LIN {X 0,Y 450.056,Z 1227.02,A -85,B 0,C 180,E1 22125.46,E2 22125.46} C_VEL
LIN {X 0,Y 451.314,Z 1216.532,A -85,B 0,C 180,E1 22122.995,E2 22122.995} C_VEL
LIN {X 0,Y 453.016,Z 1203.981,A -85,B 0,C 180,E1 22120.532,E2 22120.532} C_VEL
LIN {X 0,Y 454.944,Z 1190.743,A -85,B 0,C 180,E1 22118.331,E2 22118.331} C_VEL
LIN {X 0,Y 457.28,Z 1175.115,A -85,B 0,C 180,E1 22116.139,E2 22116.139} C_VEL
LIN {X 0,Y 459.71,Z 1158.959,A -85,B 0,C 180,E1 22114.214,E2 22114.214} C_VEL
LIN {X 0,Y 462.395,Z 1140.754,A -85,B 0,C 180,E1 22112.365,E2 22112.365} C_VEL
LIN {X 0,Y 464.992,Z 1122.424,A -85,B 0,C 180,E1 22110.782,E2 22110.782} C_VEL
LIN {X 0,Y 467.714,Z 1101.621,A -85,B 0,C 180,E1 22109.273,E2 22109.273} C_VEL
LIN {X 0,Y 470.333,Z 1079.541,A -85,B 0,C 180,E1 22107.966,E2 22107.966} C_VEL
LIN {X 0,Y 472.543,Z 1057.663,A -85,B 0,C 180,E1 22106.923,E2 22106.923} C_VEL
LIN {X 0,Y 474.461,Z 1035.079,A -85,B 0,C 180,E1 22106.08,E2 22106.08} C_VEL
LIN {X 0,Y 476.032,Z 1011.751,A -85,B 0,C 180,E1 22105.437,E2 22105.437} C_VEL
LIN {X 0,Y 488.439,Z 758.371,A -85,B 0,C 180,E1 22100.652,E2 22100.652} C_VEL
LIN {X 0,Y 471.567,Z 725.378,A -85,B 0,C 180,E1 22098.484,E2 22098.484} C_VEL
LIN {X 0,Y 462.172,Z 707.758,A -85,B 0,C 180,E1 22097.175,E2 22097.175} C_VEL
LIN {X 0,Y 454.225,Z 686.767,A -85,B 0,C 180,E1 22094.078,E2 22094.078} C_VEL
LIN {X 0,Y 450.292,Z 676.573,A -85,B 0,C 180,E1 22092.505,E2 22092.505} C_VEL
LIN {X 0,Y 450.29,Z 676.583,A -85,B 0,C 180,E1 22088.793,E2 22088.793} C_VEL
LIN {X 0,Y 450.29,Z 676.576,A -85,B 0,C 180,E1 22084.977,E2 22084.977} C_VEL
LIN {X 0,Y 450.301,Z 676.568,A -85,B 0,C 180,E1 22081.252,E2 22081.252} C_VEL
LIN {X 0,Y 450.289,Z 676.577,A -85,B 0,C 180,E1 22077.51,E2 22077.51} C_VEL
LIN {X 0,Y 450.301,Z 676.576,A -85,B 0,C 180,E1 22073.816,E2 22073.816} C_VEL
LIN {X 0,Y 450.302,Z 676.577,A -85,B 0,C 180,E1 22069.998,E2 22069.998} C_VEL
LIN {X 0,Y 450.288,Z 676.578,A -85,B 0,C 180,E1 22066.249,E2 22066.249} C_VEL
LIN {X 0,Y 450.3,Z 676.565,A -85,B 0,C 180,E1 22062.57,E2 22062.57} C_VEL
LIN {X 0,Y 450.284,Z 676.564,A -85,B 0,C 180,E1 22058.815,E2 22058.815} C_VEL
LIN {X 0,Y 450.291,Z 676.573,A -85,B 0,C 180,E1 22055.097,E2 22055.097} C_VEL
LIN {X 0,Y 450.29,Z 676.577,A -85,B 0,C 180,E1 22051.274,E2 22051.274} C_VEL
LIN {X 0,Y 450.289,Z 676.578,A -85,B 0,C 180,E1 22047.584,E2 22047.584} C_VEL
LIN {X 0,Y 450.296,Z 676.578,A -85,B 0,C 180,E1 22043.883,E2 22043.883} C_VEL
LIN {X 0,Y 450.289,Z 676.58,A -85,B 0,C 180,E1 22040.157,E2 22040.157} C_VEL
LIN {X 0,Y 450.288,Z 676.568,A -85,B 0,C 180,E1 22038.847,E2 22038.847} C_VEL
LIN {X 0,Y 449.316,Z 676.698,A -85,B 0,C 180,E1 22037.866,E2 22037.866} C_VEL
LIN {X 0,Y 442.815,Z 677.506,A -85,B 0,C 180,E1 22035.035,E2 22035.035} C_VEL
LIN {X 0,Y 442.36,Z 677.568,A -85,B 0,C 180,E1 22034.387,E2 22034.387} C_VEL
LIN {X 0,Y 442.357,Z 677.564,A -85,B 0,C 180,E1 22030.595,E2 22030.595} C_VEL
LIN {X 0,Y 442.355,Z 677.564,A -85,B 0,C 180,E1 22026.842,E2 22026.842} C_VEL
LIN {X 0,Y 442.362,Z 677.562,A -85,B 0,C 180,E1 22023.126,E2 22023.126} C_VEL
LIN {X 0,Y 442.352,Z 677.568,A -85,B 0,C 180,E1 22019.282,E2 22019.282} C_VEL
LIN {X 0,Y 442.377,Z 677.726,A -85,B 0,C 180,E1 22019.086,E2 22019.086} C_VEL
LIN {X 0,Y 443.743,Z 681.144,A -85,B 0,C 180,E1 22018.485,E2 22018.485} C_VEL
LIN {X 0,Y 450.868,Z 697.83,A -85,B 0,C 180,E1 22015.565,E2 22015.565} C_VEL
LIN {X 0,Y 458.461,Z 716.626,A -85,B 0,C 180,E1 22012.522,E2 22012.522} C_VEL
LIN {X 0,Y 466.093,Z 737.615,A -85,B 0,C 180,E1 22009.414,E2 22009.414} C_VEL
LIN {X 0,Y 472.641,Z 757.701,A -85,B 0,C 180,E1 22006.671,E2 22006.671} C_VEL
LIN {X 0,Y 467.674,Z 797.424,A -85,B 0,C 180,E1 22003.002,E2 22003.002} C_VEL
LIN {X 0,Y 462.803,Z 839.96,A -85,B 0,C 180,E1 21999.115,E2 21999.115} C_VEL
LIN {X 0,Y 458.303,Z 884.233,A -85,B 0,C 180,E1 21995.105,E2 21995.105} C_VEL
LIN {X 0,Y 455.719,Z 913.64,A -85,B 0,C 180,E1 21992.499,E2 21992.499} C_VEL
LIN {X 0,Y 456.506,Z 925.556,A -85,B 0,C 180,E1 21992.153,E2 21992.153} C_VEL
LIN {X 0,Y 451.281,Z 1032.151,A -85,B 0,C 180,E1 21989.514,E2 21989.514} C_VEL
LIN {X 0,Y 450.142,Z 1064.631,A -85,B 0,C 180,E1 21988.597,E2 21988.597} C_VEL
LIN {X 0,Y 449.375,Z 1081.923,A -85,B 0,C 180,E1 21987.857,E2 21987.857} C_VEL
LIN {X 0,Y 448.364,Z 1098.592,A -85,B 0,C 180,E1 21986.876,E2 21986.876} C_VEL
LIN {X 0,Y 447.221,Z 1113.837,A -85,B 0,C 180,E1 21985.713,E2 21985.713} C_VEL
LIN {X 0,Y 446.029,Z 1128.635,A -85,B 0,C 180,E1 21984.291,E2 21984.291} C_VEL
LIN {X 0,Y 444.836,Z 1141.996,A -85,B 0,C 180,E1 21982.674,E2 21982.674} C_VEL
LIN {X 0,Y 443.812,Z 1153.261,A -85,B 0,C 180,E1 21980.991,E2 21980.991} C_VEL
LIN {X 0,Y 442.868,Z 1164.02,A -85,B 0,C 180,E1 21978.973,E2 21978.973} C_VEL
LIN {X 0,Y 442.222,Z 1172.371,A -85,B 0,C 180,E1 21976.958,E2 21976.958} C_VEL
LIN {X 0,Y 441.818,Z 1178.872,A -85,B 0,C 180,E1 21974.915,E2 21974.915} C_VEL
LIN {X 0,Y 441.638,Z 1183.6,A -85,B 0,C 180,E1 21972.819,E2 21972.819} C_VEL
LIN {X 0,Y 441.67,Z 1186.819,A -85,B 0,C 180,E1 21970.566,E2 21970.566} C_VEL
LIN {X 0,Y 441.926,Z 1188.049,A -85,B 0,C 180,E1 21968.326,E2 21968.326} C_VEL
LIN {X 0,Y 442.395,Z 1187.557,A -85,B 0,C 180,E1 21966.228,E2 21966.228} C_VEL
LIN {X 0,Y 443.192,Z 1185.187,A -85,B 0,C 180,E1 21964.011,E2 21964.011} C_VEL
LIN {X 0,Y 444.276,Z 1181.299,A -85,B 0,C 180,E1 21961.935,E2 21961.935} C_VEL
LIN {X 0,Y 445.808,Z 1175.142,A -85,B 0,C 180,E1 21959.743,E2 21959.743} C_VEL
LIN {X 0,Y 447.557,Z 1167.915,A -85,B 0,C 180,E1 21957.823,E2 21957.823} C_VEL
LIN {X 0,Y 449.67,Z 1158.688,A -85,B 0,C 180,E1 21955.92,E2 21955.92} C_VEL
LIN {X 0,Y 451.78,Z 1148.729,A -85,B 0,C 180,E1 21954.284,E2 21954.284} C_VEL
LIN {X 0,Y 454.277,Z 1136.036,A -85,B 0,C 180,E1 21952.602,E2 21952.602} C_VEL
LIN {X 0,Y 456.731,Z 1121.995,A -85,B 0,C 180,E1 21951.121,E2 21951.121} C_VEL
LIN {X 0,Y 458.851,Z 1108.131,A -85,B 0,C 180,E1 21949.96,E2 21949.96} C_VEL
LIN {X 0,Y 460.981,Z 1091.626,A -85,B 0,C 180,E1 21948.869,E2 21948.869} C_VEL
LIN {X 0,Y 462.692,Z 1074.772,A -85,B 0,C 180,E1 21948.026,E2 21948.026} C_VEL
LIN {X 0,Y 466.759,Z 1039.48,A -85,B 0,C 180,E1 21946.627,E2 21946.627} C_VEL
LIN {X 0,Y 474.203,Z 984.707,A -85,B 0,C 180,E1 21944.726,E2 21944.726} C_VEL
LIN {X 0,Y 479.772,Z 939.46,A -85,B 0,C 180,E1 21943.332,E2 21943.332} C_VEL
LIN {X 0,Y 479.663,Z 936.85,A -85,B 0,C 180,E1 21943.157,E2 21943.157} C_VEL
LIN {X 0,Y 489.104,Z 900.674,A -85,B 0,C 180,E1 21939.288,E2 21939.288} C_VEL
LIN {X 0,Y 499.739,Z 867.838,A -85,B 0,C 180,E1 21935.659,E2 21935.659} C_VEL
LIN {X 0,Y 511.957,Z 837.578,A -85,B 0,C 180,E1 21932.174,E2 21932.174} C_VEL
LIN {X 0,Y 521.645,Z 817.739,A -85,B 0,C 180,E1 21929.791,E2 21929.791} C_VEL
LIN {X 0,Y 522.316,Z 814.236,A -85,B 0,C 180,E1 21928.105,E2 21928.105} C_VEL
LIN {X 0,Y 522.83,Z 812.775,A -85,B 0,C 180,E1 21926.841,E2 21926.841} C_VEL
LIN {X 0,Y 523.839,Z 811.873,A -85,B 0,C 180,E1 21925.332,E2 21925.332} C_VEL
LIN {X 0,Y 523.786,Z 813.12,A -85,B 0,C 180,E1 21924.408,E2 21924.408} C_VEL
LIN {X 0,Y 511.159,Z 837.266,A -85,B 0,C 180,E1 21922.025,E2 21922.025} C_VEL
LIN {X 0,Y 502.911,Z 857.599,A -85,B 0,C 180,E1 21919.896,E2 21919.896} C_VEL
LIN {X 0,Y 497.203,Z 877.592,A -85,B 0,C 180,E1 21917.647,E2 21917.647} C_VEL
LIN {X 0,Y 494.543,Z 895.305,A -85,B 0,C 180,E1 21915.535,E2 21915.535} C_VEL
LIN {X 0,Y 494.336,Z 913.318,A -85,B 0,C 180,E1 21913.266,E2 21913.266} C_VEL
LIN {X 0,Y 496.692,Z 929.505,A -85,B 0,C 180,E1 21911.157,E2 21911.157} C_VEL
LIN {X 0,Y 501.231,Z 945.016,A -85,B 0,C 180,E1 21909.095,E2 21909.095} C_VEL
LIN {X 0,Y 488.403,Z 970.998,A -85,B 0,C 180,E1 21908.038,E2 21908.038} C_VEL
LIN {X 0,Y 478.774,Z 994.4,A -85,B 0,C 180,E1 21906.916,E2 21906.916} C_VEL
LIN {X 0,Y 474.737,Z 1026.804,A -85,B 0,C 180,E1 21906.44,E2 21906.44} C_VEL
LIN {X 0,Y 472.39,Z 1050.839,A -85,B 0,C 180,E1 21905.821,E2 21905.821} C_VEL
LIN {X 0,Y 469.098,Z 1076.984,A -85,B 0,C 180,E1 21904.909,E2 21904.909} C_VEL
LIN {X 0,Y 465.898,Z 1098.995,A -85,B 0,C 180,E1 21903.915,E2 21903.915} C_VEL
LIN {X 0,Y 462.099,Z 1123.392,A -85,B 0,C 180,E1 21902.525,E2 21902.525} C_VEL
LIN {X 0,Y 458.733,Z 1143.969,A -85,B 0,C 180,E1 21901.101,E2 21901.101} C_VEL
LIN {X 0,Y 453.603,Z 1177.436,A -85,B 0,C 180,E1 21898.359,E2 21898.359} C_VEL
LIN {X 0,Y 450.76,Z 1196.691,A -85,B 0,C 180,E1 21896.476,E2 21896.476} C_VEL
LIN {X 0,Y 448.232,Z 1213.866,A -85,B 0,C 180,E1 21894.474,E2 21894.474} C_VEL
LIN {X 0,Y 446.026,Z 1229.04,A -85,B 0,C 180,E1 21892.4,E2 21892.4} C_VEL
LIN {X 0,Y 444.101,Z 1243.186,A -85,B 0,C 180,E1 21890.136,E2 21890.136} C_VEL
LIN {X 0,Y 442.582,Z 1255.81,A -85,B 0,C 180,E1 21887.756,E2 21887.756} C_VEL
LIN {X 0,Y 441.424,Z 1266.903,A -85,B 0,C 180,E1 21885.232,E2 21885.232} C_VEL
LIN {X 0,Y 440.697,Z 1276.161,A -85,B 0,C 180,E1 21882.676,E2 21882.676} C_VEL
LIN {X 0,Y 440.308,Z 1283.784,A -85,B 0,C 180,E1 21880.068,E2 21880.068} C_VEL
LIN {X 0,Y 440.178,Z 1289.391,A -85,B 0,C 180,E1 21877.569,E2 21877.569} C_VEL
LIN {X 0,Y 440.187,Z 1293.587,A -85,B 0,C 180,E1 21874.95,E2 21874.95} C_VEL
LIN {X 0,Y 440.235,Z 1296.109,A -85,B 0,C 180,E1 21872.472,E2 21872.472} C_VEL
LIN {X 0,Y 440.268,Z 1297.032,A -85,B 0,C 180,E1 21869.998,E2 21869.998} C_VEL
LIN {X 0,Y 440.212,Z 1296.537,A -85,B 0,C 180,E1 21867.395,E2 21867.395} C_VEL
LIN {X 0,Y 440.144,Z 1294.495,A -85,B 0,C 180,E1 21864.915,E2 21864.915} C_VEL
LIN {X 0,Y 440.148,Z 1290.595,A -85,B 0,C 180,E1 21862.164,E2 21862.164} C_VEL
LIN {X 0,Y 440.341,Z 1285.146,A -85,B 0,C 180,E1 21859.491,E2 21859.491} C_VEL
LIN {X 0,Y 440.893,Z 1277.648,A -85,B 0,C 180,E1 21856.757,E2 21856.757} C_VEL
LIN {X 0,Y 441.861,Z 1268.533,A -85,B 0,C 180,E1 21854.1,E2 21854.1} C_VEL
LIN {X 0,Y 443.288,Z 1258.134,A -85,B 0,C 180,E1 21851.59,E2 21851.59} C_VEL
LIN {X 0,Y 445.269,Z 1245.64,A -85,B 0,C 180,E1 21849.079,E2 21849.079} C_VEL
LIN {X 0,Y 447.716,Z 1231.692,A -85,B 0,C 180,E1 21846.714,E2 21846.714} C_VEL
LIN {X 0,Y 450.8,Z 1215.453,A -85,B 0,C 180,E1 21844.371,E2 21844.371} C_VEL
LIN {X 0,Y 454.225,Z 1198.101,A -85,B 0,C 180,E1 21842.243,E2 21842.243} C_VEL
LIN {X 0,Y 457.98,Z 1179.391,A -85,B 0,C 180,E1 21840.289,E2 21840.289} C_VEL
LIN {X 0,Y 462.201,Z 1158.237,A -85,B 0,C 180,E1 21838.43,E2 21838.43} C_VEL
LIN {X 0,Y 466.546,Z 1136.041,A -85,B 0,C 180,E1 21836.797,E2 21836.797} C_VEL
LIN {X 0,Y 470.757,Z 1113.889,A -85,B 0,C 180,E1 21835.45,E2 21835.45} C_VEL
LIN {X 0,Y 475.07,Z 1090.125,A -85,B 0,C 180,E1 21834.262,E2 21834.262} C_VEL
LIN {X 0,Y 479.303,Z 1065.271,A -85,B 0,C 180,E1 21833.286,E2 21833.286} C_VEL
LIN {X 0,Y 483.325,Z 1037.764,A -85,B 0,C 180,E1 21832.445,E2 21832.445} C_VEL
LIN {X 0,Y 486.658,Z 1015.568,A -85,B 0,C 180,E1 21831.951,E2 21831.951} C_VEL
LIN {X 0,Y 492.888,Z 982.261,A -85,B 0,C 180,E1 21831.411,E2 21831.411} C_VEL
LIN {X 0,Y 499.024,Z 954.26,A -85,B 0,C 180,E1 21831.118,E2 21831.118} C_VEL
LIN {X 0,Y 501.49,Z 943.396,A -85,B 0,C 180,E1 21831.019,E2 21831.019} C_VEL
LIN {X 0,Y 498.054,Z 928.988,A -85,B 0,C 180,E1 21829.189,E2 21829.189} C_VEL
LIN {X 0,Y 497.038,Z 917.484,A -85,B 0,C 180,E1 21827.693,E2 21827.693} C_VEL
LIN {X 0,Y 497.581,Z 906.994,A -85,B 0,C 180,E1 21826.402,E2 21826.402} C_VEL
LIN {X 0,Y 499.538,Z 895.357,A -85,B 0,C 180,E1 21824.944,E2 21824.944} C_VEL
LIN {X 0,Y 502.528,Z 884.79,A -85,B 0,C 180,E1 21823.757,E2 21823.757} C_VEL
LIN {X 0,Y 506.992,Z 873.197,A -85,B 0,C 180,E1 21822.425,E2 21822.425} C_VEL
LIN {X 0,Y 510.787,Z 864.66,A -85,B 0,C 180,E1 21821.584,E2 21821.584} C_VEL
LIN {X 0,Y 498.036,Z 933.263,A -85,B 0,C 180,E1 21819.708,E2 21819.708} C_VEL
LIN {X 0,Y 488.405,Z 996.354,A -85,B 0,C 180,E1 21818.004,E2 21818.004} C_VEL
LIN {X 0,Y 483.779,Z 1031.006,A -85,B 0,C 180,E1 21817.02,E2 21817.02} C_VEL
LIN {X 0,Y 480.204,Z 1054.828,A -85,B 0,C 180,E1 21816.105,E2 21816.105} C_VEL
LIN {X 0,Y 476.468,Z 1077.16,A -85,B 0,C 180,E1 21815.027,E2 21815.027} C_VEL
LIN {X 0,Y 472.331,Z 1099.651,A -85,B 0,C 180,E1 21813.686,E2 21813.686} C_VEL
LIN {X 0,Y 468.084,Z 1121.13,A -85,B 0,C 180,E1 21812.134,E2 21812.134} C_VEL
LIN {X 0,Y 463.799,Z 1141.476,A -85,B 0,C 180,E1 21810.368,E2 21810.368} C_VEL
LIN {X 0,Y 459.71,Z 1160.043,A -85,B 0,C 180,E1 21808.446,E2 21808.446} C_VEL
LIN {X 0,Y 455.964,Z 1176.51,A -85,B 0,C 180,E1 21806.434,E2 21806.434} C_VEL
LIN {X 0,Y 452.524,Z 1191.573,A -85,B 0,C 180,E1 21804.267,E2 21804.267} C_VEL
LIN {X 0,Y 449.427,Z 1205.245,A -85,B 0,C 180,E1 21801.948,E2 21801.948} C_VEL
LIN {X 0,Y 446.744,Z 1217.484,A -85,B 0,C 180,E1 21799.481,E2 21799.481} C_VEL
LIN {X 0,Y 444.509,Z 1228.139,A -85,B 0,C 180,E1 21796.869,E2 21796.869} C_VEL
LIN {X 0,Y 442.835,Z 1236.857,A -85,B 0,C 180,E1 21794.248,E2 21794.248} C_VEL
LIN {X 0,Y 441.629,Z 1244.145,A -85,B 0,C 180,E1 21791.493,E2 21791.493} C_VEL
LIN {X 0,Y 440.859,Z 1249.657,A -85,B 0,C 180,E1 21788.741,E2 21788.741} C_VEL
LIN {X 0,Y 440.421,Z 1253.357,A -85,B 0,C 180,E1 21785.995,E2 21785.995} C_VEL
LIN {X 0,Y 440.195,Z 1255.428,A -85,B 0,C 180,E1 21783.255,E2 21783.255} C_VEL
LIN {X 0,Y 440.127,Z 1255.953,A -85,B 0,C 180,E1 21780.651,E2 21780.651} C_VEL
LIN {X 0,Y 440.098,Z 1254.877,A -85,B 0,C 180,E1 21778.047,E2 21778.047} C_VEL
LIN {X 0,Y 440.145,Z 1252.176,A -85,B 0,C 180,E1 21775.309,E2 21775.309} C_VEL
LIN {X 0,Y 440.324,Z 1248.078,A -85,B 0,C 180,E1 21772.694,E2 21772.694} C_VEL
LIN {X 0,Y 440.684,Z 1242.233,A -85,B 0,C 180,E1 21770.07,E2 21770.07} C_VEL
LIN {X 0,Y 441.337,Z 1234.695,A -85,B 0,C 180,E1 21767.438,E2 21767.438} C_VEL
LIN {X 0,Y 442.336,Z 1225.49,A -85,B 0,C 180,E1 21764.849,E2 21764.849} C_VEL
LIN {X 0,Y 443.756,Z 1214.389,A -85,B 0,C 180,E1 21762.291,E2 21762.291} C_VEL
LIN {X 0,Y 445.497,Z 1201.996,A -85,B 0,C 180,E1 21759.916,E2 21759.916} C_VEL
LIN {X 0,Y 447.593,Z 1188.047,A -85,B 0,C 180,E1 21757.647,E2 21757.647} C_VEL
LIN {X 0,Y 449.987,Z 1172.681,A -85,B 0,C 180,E1 21755.518,E2 21755.518} C_VEL
LIN {X 0,Y 452.643,Z 1155.548,A -85,B 0,C 180,E1 21753.499,E2 21753.499} C_VEL
LIN {X 0,Y 455.388,Z 1137.286,A -85,B 0,C 180,E1 21751.688,E2 21751.688} C_VEL
LIN {X 0,Y 458.1,Z 1118.169,A -85,B 0,C 180,E1 21750.083,E2 21750.083} C_VEL
LIN {X 0,Y 460.848,Z 1097.369,A -85,B 0,C 180,E1 21748.619,E2 21748.619} C_VEL
LIN {X 0,Y 463.351,Z 1076.315,A -85,B 0,C 180,E1 21747.396,E2 21747.396} C_VEL
LIN {X 0,Y 465.634,Z 1054.147,A -85,B 0,C 180,E1 21746.356,E2 21746.356} C_VEL
LIN {X 0,Y 467.579,Z 1031.116,A -85,B 0,C 180,E1 21745.527,E2 21745.527} C_VEL
LIN {X 0,Y 469.041,Z 1008.426,A -85,B 0,C 180,E1 21744.93,E2 21744.93} C_VEL
LIN {X 0,Y 481.668,Z 761.074,A -85,B 0,C 180,E1 21740.183,E2 21740.183} C_VEL
LIN {X 0,Y 465.208,Z 728.878,A -85,B 0,C 180,E1 21738.023,E2 21738.023} C_VEL
LIN {X 0,Y 454.223,Z 708.49,A -85,B 0,C 180,E1 21736.498,E2 21736.498} C_VEL
LIN {X 0,Y 446.291,Z 687.68,A -85,B 0,C 180,E1 21733.371,E2 21733.371} C_VEL
LIN {X 0,Y 442.359,Z 677.565,A -85,B 0,C 180,E1 21731.762,E2 21731.762} C_VEL
LIN {X 0,Y 442.36,Z 677.564,A -85,B 0,C 180,E1 21727.92,E2 21727.92} C_VEL
LIN {X 0,Y 442.354,Z 677.558,A -85,B 0,C 180,E1 21724.177,E2 21724.177} C_VEL
LIN {X 0,Y 442.356,Z 677.557,A -85,B 0,C 180,E1 21720.421,E2 21720.421} C_VEL
LIN {X 0,Y 442.353,Z 677.566,A -85,B 0,C 180,E1 21716.733,E2 21716.733} C_VEL
LIN {X 0,Y 442.366,Z 677.566,A -85,B 0,C 180,E1 21713.02,E2 21713.02} C_VEL
LIN {X 0,Y 442.35,Z 677.563,A -85,B 0,C 180,E1 21709.271,E2 21709.271} C_VEL
LIN {X 0,Y 442.355,Z 677.565,A -85,B 0,C 180,E1 21705.471,E2 21705.471} C_VEL
LIN {X 0,Y 442.351,Z 677.561,A -85,B 0,C 180,E1 21701.74,E2 21701.74} C_VEL
LIN {X 0,Y 442.362,Z 677.551,A -85,B 0,C 180,E1 21697.927,E2 21697.927} C_VEL
LIN {X 0,Y 442.349,Z 677.556,A -85,B 0,C 180,E1 21694.28,E2 21694.28} C_VEL
LIN {X 0,Y 442.358,Z 677.558,A -85,B 0,C 180,E1 21690.52,E2 21690.52} C_VEL
LIN {X 0,Y 442.351,Z 677.56,A -85,B 0,C 180,E1 21686.762,E2 21686.762} C_VEL
LIN {X 0,Y 442.354,Z 677.559,A -85,B 0,C 180,E1 21682.991,E2 21682.991} C_VEL
LIN {X 0,Y 442.347,Z 677.558,A -85,B 0,C 180,E1 21679.188,E2 21679.188} C_VEL
LIN {X 0,Y 442.368,Z 677.558,A -85,B 0,C 180,E1 21675.472,E2 21675.472} C_VEL
LIN {X 0,Y 442.36,Z 677.568,A -85,B 0,C 180,E1 21674.387,E2 21674.387} C_VEL
LIN {X 0,Y 441.352,Z 677.703,A -85,B 0,C 180,E1 21673.389,E2 21673.389} C_VEL
LIN {X 0,Y 434.853,Z 678.499,A -85,B 0,C 180,E1 21670.507,E2 21670.507} C_VEL
LIN {X 0,Y 434.412,Z 678.55,A -85,B 0,C 180,E1 21669.846,E2 21669.846} C_VEL
LIN {X 0,Y 434.42,Z 678.557,A -85,B 0,C 180,E1 21666.031,E2 21666.031} C_VEL
LIN {X 0,Y 434.421,Z 678.551,A -85,B 0,C 180,E1 21662.147,E2 21662.147} C_VEL
LIN {X 0,Y 434.434,Z 678.618,A -85,B 0,C 180,E1 21660.039,E2 21660.039} C_VEL
LIN {X 0,Y 435.836,Z 682.213,A -85,B 0,C 180,E1 21659.385,E2 21659.385} C_VEL
LIN {X 0,Y 442.612,Z 697.837,A -85,B 0,C 180,E1 21656.553,E2 21656.553} C_VEL
LIN {X 0,Y 449.79,Z 715.531,A -85,B 0,C 180,E1 21653.594,E2 21653.594} C_VEL
LIN {X 0,Y 457.241,Z 735.445,A -85,B 0,C 180,E1 21650.528,E2 21650.528} C_VEL
LIN {X 0,Y 464.319,Z 756.568,A -85,B 0,C 180,E1 21647.541,E2 21647.541} C_VEL
LIN {X 0,Y 465.547,Z 760.574,A -85,B 0,C 180,E1 21647.001,E2 21647.001} C_VEL
LIN {X 0,Y 460.466,Z 799.942,A -85,B 0,C 180,E1 21643.329,E2 21643.329} C_VEL
LIN {X 0,Y 455.418,Z 842.649,A -85,B 0,C 180,E1 21639.384,E2 21639.384} C_VEL
LIN {X 0,Y 450.821,Z 886.432,A -85,B 0,C 180,E1 21635.372,E2 21635.372} C_VEL
LIN {X 0,Y 448.282,Z 914.377,A -85,B 0,C 180,E1 21632.867,E2 21632.867} C_VEL
LIN {X 0,Y 449.028,Z 926.332,A -85,B 0,C 180,E1 21632.508,E2 21632.508} C_VEL
LIN {X 0,Y 443.831,Z 1028.572,A -85,B 0,C 180,E1 21629.921,E2 21629.921} C_VEL
LIN {X 0,Y 442.45,Z 1064.95,A -85,B 0,C 180,E1 21628.876,E2 21628.876} C_VEL
LIN {X 0,Y 441.667,Z 1082.248,A -85,B 0,C 180,E1 21628.129,E2 21628.129} C_VEL
LIN {X 0,Y 440.625,Z 1098.826,A -85,B 0,C 180,E1 21627.137,E2 21627.137} C_VEL
LIN {X 0,Y 439.463,Z 1113.913,A -85,B 0,C 180,E1 21625.976,E2 21625.976} C_VEL
LIN {X 0,Y 438.231,Z 1128.717,A -85,B 0,C 180,E1 21624.536,E2 21624.536} C_VEL
LIN {X 0,Y 437.042,Z 1141.718,A -85,B 0,C 180,E1 21622.96,E2 21622.96} C_VEL
LIN {X 0,Y 435.975,Z 1153.218,A -85,B 0,C 180,E1 21621.246,E2 21621.246} C_VEL
LIN {X 0,Y 435.093,Z 1162.863,A -85,B 0,C 180,E1 21619.465,E2 21619.465} C_VEL
LIN {X 0,Y 434.381,Z 1171.744,A -85,B 0,C 180,E1 21617.412,E2 21617.412} C_VEL
LIN {X 0,Y 433.926,Z 1178.508,A -85,B 0,C 180,E1 21615.367,E2 21615.367} C_VEL
LIN {X 0,Y 433.699,Z 1183.794,A -85,B 0,C 180,E1 21613.194,E2 21613.194} C_VEL
LIN {X 0,Y 433.694,Z 1187.191,A -85,B 0,C 180,E1 21611.032,E2 21611.032} C_VEL
LIN {X 0,Y 433.933,Z 1188.99,A -85,B 0,C 180,E1 21608.707,E2 21608.707} C_VEL
LIN {X 0,Y 434.4,Z 1188.827,A -85,B 0,C 180,E1 21606.476,E2 21606.476} C_VEL
LIN {X 0,Y 435.2,Z 1186.91,A -85,B 0,C 180,E1 21604.216,E2 21604.216} C_VEL
LIN {X 0,Y 436.446,Z 1182.789,A -85,B 0,C 180,E1 21601.838,E2 21601.838} C_VEL
LIN {X 0,Y 437.951,Z 1177.292,A -85,B 0,C 180,E1 21599.738,E2 21599.738} C_VEL
LIN {X 0,Y 439.889,Z 1169.908,A -85,B 0,C 180,E1 21597.655,E2 21597.655} C_VEL
LIN {X 0,Y 442.081,Z 1160.89,A -85,B 0,C 180,E1 21595.72,E2 21595.72} C_VEL
LIN {X 0,Y 444.476,Z 1150.465,A -85,B 0,C 180,E1 21593.931,E2 21593.931} C_VEL
LIN {X 0,Y 447.107,Z 1138.01,A -85,B 0,C 180,E1 21592.224,E2 21592.224} C_VEL
LIN {X 0,Y 449.555,Z 1124.833,A -85,B 0,C 180,E1 21590.785,E2 21590.785} C_VEL
LIN {X 0,Y 451.917,Z 1110.832,A -85,B 0,C 180,E1 21589.547,E2 21589.547} C_VEL
LIN {X 0,Y 454.173,Z 1095.021,A -85,B 0,C 180,E1 21588.443,E2 21588.443} C_VEL
LIN {X 0,Y 455.954,Z 1078.953,A -85,B 0,C 180,E1 21587.59,E2 21587.59} C_VEL
LIN {X 0,Y 459.956,Z 1045.813,A -85,B 0,C 180,E1 21586.197,E2 21586.197} C_VEL
LIN {X 0,Y 468.298,Z 988.208,A -85,B 0,C 180,E1 21584.119,E2 21584.119} C_VEL
LIN {X 0,Y 474.305,Z 941.492,A -85,B 0,C 180,E1 21582.66,E2 21582.66} C_VEL
LIN {X 0,Y 474.187,Z 938.407,A -85,B 0,C 180,E1 21582.45,E2 21582.45} C_VEL
LIN {X 0,Y 483.685,Z 904.18,A -85,B 0,C 180,E1 21578.728,E2 21578.728} C_VEL
LIN {X 0,Y 495.003,Z 871.247,A -85,B 0,C 180,E1 21575.028,E2 21575.028} C_VEL
LIN {X 0,Y 507.35,Z 842.267,A -85,B 0,C 180,E1 21571.643,E2 21571.643} C_VEL
LIN {X 0,Y 517.091,Z 823.34,A -85,B 0,C 180,E1 21569.339,E2 21569.339} C_VEL
LIN {X 0,Y 517.922,Z 820.031,A -85,B 0,C 180,E1 21567.525,E2 21567.525} C_VEL
LIN {X 0,Y 519.259,Z 818.526,A -85,B 0,C 180,E1 21565.305,E2 21565.305} C_VEL
LIN {X 0,Y 519.194,Z 819.101,A -85,B 0,C 180,E1 21564.877,E2 21564.877} C_VEL
LIN {X 0,Y 506.191,Z 843.075,A -85,B 0,C 180,E1 21562.472,E2 21562.472} C_VEL
LIN {X 0,Y 497.568,Z 863.437,A -85,B 0,C 180,E1 21560.28,E2 21560.28} C_VEL
LIN {X 0,Y 491.782,Z 883.1,A -85,B 0,C 180,E1 21558.016,E2 21558.016} C_VEL
LIN {X 0,Y 488.921,Z 900.513,A -85,B 0,C 180,E1 21555.872,E2 21555.872} C_VEL
LIN {X 0,Y 488.536,Z 917.775,A -85,B 0,C 180,E1 21553.646,E2 21553.646} C_VEL
LIN {X 0,Y 490.708,Z 934.335,A -85,B 0,C 180,E1 21551.422,E2 21551.422} C_VEL
LIN {X 0,Y 494.318,Z 947.396,A -85,B 0,C 180,E1 21549.64,E2 21549.64} C_VEL
LIN {X 0,Y 483.213,Z 969.576,A -85,B 0,C 180,E1 21548.749,E2 21548.749} C_VEL
LIN {X 0,Y 473.292,Z 993.014,A -85,B 0,C 180,E1 21547.617,E2 21547.617} C_VEL
LIN {X 0,Y 468.929,Z 1026.776,A -85,B 0,C 180,E1 21547.109,E2 21547.109} C_VEL
LIN {X 0,Y 466.3,Z 1051.355,A -85,B 0,C 180,E1 21546.451,E2 21546.451} C_VEL
LIN {X 0,Y 463.064,Z 1075.696,A -85,B 0,C 180,E1 21545.584,E2 21545.584} C_VEL
LIN {X 0,Y 459.691,Z 1097.445,A -85,B 0,C 180,E1 21544.588,E2 21544.588} C_VEL
LIN {X 0,Y 455.844,Z 1120.852,A -85,B 0,C 180,E1 21543.253,E2 21543.253} C_VEL
LIN {X 0,Y 452.113,Z 1142.301,A -85,B 0,C 180,E1 21541.757,E2 21541.757} C_VEL
LIN {X 0,Y 448.436,Z 1162.901,A -85,B 0,C 180,E1 21540.035,E2 21540.035} C_VEL
LIN {X 0,Y 443.615,Z 1192.753,A -85,B 0,C 180,E1 21537.154,E2 21537.154} C_VEL
LIN {X 0,Y 440.965,Z 1210.228,A -85,B 0,C 180,E1 21535.158,E2 21535.158} C_VEL
LIN {X 0,Y 438.638,Z 1225.751,A -85,B 0,C 180,E1 21533.082,E2 21533.082} C_VEL
LIN {X 0,Y 436.581,Z 1240.312,A -85,B 0,C 180,E1 21530.791,E2 21530.791} C_VEL
LIN {X 0,Y 434.977,Z 1252.62,A -85,B 0,C 180,E1 21528.493,E2 21528.493} C_VEL
LIN {X 0,Y 433.681,Z 1264.259,A -85,B 0,C 180,E1 21525.922,E2 21525.922} C_VEL
LIN {X 0,Y 432.856,Z 1273.905,A -85,B 0,C 180,E1 21523.354,E2 21523.354} C_VEL
LIN {X 0,Y 432.375,Z 1281.623,A -85,B 0,C 180,E1 21520.794,E2 21520.794} C_VEL
LIN {X 0,Y 432.199,Z 1287.93,A -85,B 0,C 180,E1 21518.111,E2 21518.111} C_VEL
LIN {X 0,Y 432.19,Z 1292.368,A -85,B 0,C 180,E1 21515.574,E2 21515.574} C_VEL
LIN {X 0,Y 432.245,Z 1295.146,A -85,B 0,C 180,E1 21513.048,E2 21513.048} C_VEL
LIN {X 0,Y 432.268,Z 1296.563,A -85,B 0,C 180,E1 21510.396,E2 21510.396} C_VEL
LIN {X 0,Y 432.232,Z 1296.379,A -85,B 0,C 180,E1 21507.948,E2 21507.948} C_VEL
LIN {X 0,Y 432.154,Z 1294.578,A -85,B 0,C 180,E1 21505.22,E2 21505.22} C_VEL
LIN {X 0,Y 432.15,Z 1291.241,A -85,B 0,C 180,E1 21502.554,E2 21502.554} C_VEL
LIN {X 0,Y 432.301,Z 1286.167,A -85,B 0,C 180,E1 21499.874,E2 21499.874} C_VEL
LIN {X 0,Y 432.819,Z 1279.066,A -85,B 0,C 180,E1 21497.049,E2 21497.049} C_VEL
LIN {X 0,Y 433.765,Z 1270.496,A -85,B 0,C 180,E1 21494.352,E2 21494.352} C_VEL
LIN {X 0,Y 435.266,Z 1259.877,A -85,B 0,C 180,E1 21491.655,E2 21491.655} C_VEL
LIN {X 0,Y 437.281,Z 1247.834,A -85,B 0,C 180,E1 21489.1,E2 21489.1} C_VEL
LIN {X 0,Y 439.948,Z 1233.637,A -85,B 0,C 180,E1 21486.562,E2 21486.562} C_VEL
LIN {X 0,Y 443.15,Z 1217.91,A -85,B 0,C 180,E1 21484.183,E2 21484.183} C_VEL
LIN {X 0,Y 446.907,Z 1200.062,A -85,B 0,C 180,E1 21481.902,E2 21481.902} C_VEL
LIN {X 0,Y 450.972,Z 1181.068,A -85,B 0,C 180,E1 21479.85,E2 21479.85} C_VEL
LIN {X 0,Y 455.217,Z 1161.264,A -85,B 0,C 180,E1 21478.036,E2 21478.036} C_VEL
LIN {X 0,Y 459.909,Z 1139.175,A -85,B 0,C 180,E1 21476.329,E2 21476.329} C_VEL
LIN {X 0,Y 464.759,Z 1115.822,A -85,B 0,C 180,E1 21474.84,E2 21474.84} C_VEL
LIN {X 0,Y 469.525,Z 1091.745,A -85,B 0,C 180,E1 21473.588,E2 21473.588} C_VEL
LIN {X 0,Y 474.062,Z 1067.611,A -85,B 0,C 180,E1 21472.593,E2 21472.593} C_VEL
LIN {X 0,Y 478.676,Z 1039.318,A -85,B 0,C 180,E1 21471.687,E2 21471.687} C_VEL
LIN {X 0,Y 482.202,Z 1017.384,A -85,B 0,C 180,E1 21471.174,E2 21471.174} C_VEL
LIN {X 0,Y 488.593,Z 984.475,A -85,B 0,C 180,E1 21470.623,E2 21470.623} C_VEL
LIN {X 0,Y 494.848,Z 956.41,A -85,B 0,C 180,E1 21470.313,E2 21470.313} C_VEL
LIN {X 0,Y 497.113,Z 946.703,A -85,B 0,C 180,E1 21470.227,E2 21470.227} C_VEL
LIN {X 0,Y 494.838,Z 934.347,A -85,B 0,C 180,E1 21468.606,E2 21468.606} C_VEL
LIN {X 0,Y 494.412,Z 922.645,A -85,B 0,C 180,E1 21467.052,E2 21467.052} C_VEL
LIN {X 0,Y 495.491,Z 912.358,A -85,B 0,C 180,E1 21465.757,E2 21465.757} C_VEL
LIN {X 0,Y 498.136,Z 900.7,A -85,B 0,C 180,E1 21464.279,E2 21464.279} C_VEL
LIN {X 0,Y 501.656,Z 890.22,A -85,B 0,C 180,E1 21463.091,E2 21463.091} C_VEL
LIN {X 0,Y 505.516,Z 881.377,A -85,B 0,C 180,E1 21462.022,E2 21462.022} C_VEL
LIN {X 0,Y 492.101,Z 950.377,A -85,B 0,C 180,E1 21460.108,E2 21460.108} C_VEL
LIN {X 0,Y 481.773,Z 1015.305,A -85,B 0,C 180,E1 21458.319,E2 21458.319} C_VEL
LIN {X 0,Y 478.245,Z 1038.633,A -85,B 0,C 180,E1 21457.56,E2 21457.56} C_VEL
LIN {X 0,Y 474.192,Z 1062.332,A -85,B 0,C 180,E1 21456.562,E2 21456.562} C_VEL
LIN {X 0,Y 469.904,Z 1084.987,A -85,B 0,C 180,E1 21455.365,E2 21455.365} C_VEL
LIN {X 0,Y 465.444,Z 1106.79,A -85,B 0,C 180,E1 21453.955,E2 21453.955} C_VEL
LIN {X 0,Y 460.89,Z 1127.712,A -85,B 0,C 180,E1 21452.329,E2 21452.329} C_VEL
LIN {X 0,Y 456.335,Z 1147.592,A -85,B 0,C 180,E1 21450.481,E2 21450.481} C_VEL
LIN {X 0,Y 451.872,Z 1166.301,A -85,B 0,C 180,E1 21448.408,E2 21448.408} C_VEL
LIN {X 0,Y 448.083,Z 1181.942,A -85,B 0,C 180,E1 21446.364,E2 21446.364} C_VEL
LIN {X 0,Y 444.387,Z 1197.06,A -85,B 0,C 180,E1 21444.033,E2 21444.033} C_VEL
LIN {X 0,Y 441.114,Z 1210.567,A -85,B 0,C 180,E1 21441.544,E2 21441.544} C_VEL
LIN {X 0,Y 438.443,Z 1221.909,A -85,B 0,C 180,E1 21439.033,E2 21439.033} C_VEL
LIN {X 0,Y 436.258,Z 1231.863,A -85,B 0,C 180,E1 21436.374,E2 21436.374} C_VEL
LIN {X 0,Y 434.648,Z 1239.996,A -85,B 0,C 180,E1 21433.707,E2 21433.707} C_VEL
LIN {X 0,Y 433.481,Z 1246.647,A -85,B 0,C 180,E1 21430.903,E2 21430.903} C_VEL
LIN {X 0,Y 432.787,Z 1251.274,A -85,B 0,C 180,E1 21428.236,E2 21428.236} C_VEL
LIN {X 0,Y 432.379,Z 1254.559,A -85,B 0,C 180,E1 21425.441,E2 21425.441} C_VEL
LIN {X 0,Y 432.192,Z 1256.146,A -85,B 0,C 180,E1 21422.785,E2 21422.785} C_VEL
LIN {X 0,Y 432.12,Z 1256.2,A -85,B 0,C 180,E1 21420.133,E2 21420.133} C_VEL
LIN {X 0,Y 432.107,Z 1254.844,A -85,B 0,C 180,E1 21417.48,E2 21417.48} C_VEL
LIN {X 0,Y 432.174,Z 1251.872,A -85,B 0,C 180,E1 21414.823,E2 21414.823} C_VEL
LIN {X 0,Y 432.394,Z 1247.098,A -85,B 0,C 180,E1 21412.025,E2 21412.025} C_VEL
LIN {X 0,Y 432.83,Z 1240.898,A -85,B 0,C 180,E1 21409.35,E2 21409.35} C_VEL
LIN {X 0,Y 433.6,Z 1232.863,A -85,B 0,C 180,E1 21406.667,E2 21406.667} C_VEL
LIN {X 0,Y 434.746,Z 1223.036,A -85,B 0,C 180,E1 21404.027,E2 21404.027} C_VEL
LIN {X 0,Y 436.33,Z 1211.323,A -85,B 0,C 180,E1 21401.426,E2 21401.426} C_VEL
LIN {X 0,Y 438.264,Z 1198.355,A -85,B 0,C 180,E1 21399.011,E2 21399.011} C_VEL
LIN {X 0,Y 440.533,Z 1183.928,A -85,B 0,C 180,E1 21396.738,E2 21396.738} C_VEL
LIN {X 0,Y 443.062,Z 1167.938,A -85,B 0,C 180,E1 21394.609,E2 21394.609} C_VEL
LIN {X 0,Y 445.833,Z 1150.442,A -85,B 0,C 180,E1 21392.628,E2 21392.628} C_VEL
LIN {X 0,Y 448.746,Z 1131.284,A -85,B 0,C 180,E1 21390.792,E2 21390.792} C_VEL
LIN {X 0,Y 451.534,Z 1111.928,A -85,B 0,C 180,E1 21389.228,E2 21389.228} C_VEL
LIN {X 0,Y 454.305,Z 1090.987,A -85,B 0,C 180,E1 21387.817,E2 21387.817} C_VEL
LIN {X 0,Y 456.878,Z 1068.793,A -85,B 0,C 180,E1 21386.604,E2 21386.604} C_VEL
LIN {X 0,Y 459.03,Z 1046.989,A -85,B 0,C 180,E1 21385.655,E2 21385.655} C_VEL
LIN {X 0,Y 460.908,Z 1023.435,A -85,B 0,C 180,E1 21384.868,E2 21384.868} C_VEL
LIN {X 0,Y 462.414,Z 998.384,A -85,B 0,C 180,E1 21384.279,E2 21384.279} C_VEL
LIN {X 0,Y 474.088,Z 777.34,A -85,B 0,C 180,E1 21379.961,E2 21379.961} C_VEL
LIN {X 0,Y 474.75,Z 763.422,A -85,B 0,C 180,E1 21379.68,E2 21379.68} C_VEL
LIN {X 0,Y 458.043,Z 730.762,A -85,B 0,C 180,E1 21377.434,E2 21377.434} C_VEL
LIN {X 0,Y 446.115,Z 708.779,A -85,B 0,C 180,E1 21375.735,E2 21375.735} C_VEL
LIN {X 0,Y 438.557,Z 689.045,A -85,B 0,C 180,E1 21372.711,E2 21372.711} C_VEL
LIN {X 0,Y 434.412,Z 678.561,A -85,B 0,C 180,E1 21371.046,E2 21371.046} C_VEL
LIN {X 0,Y 434.414,Z 678.548,A -85,B 0,C 180,E1 21367.213,E2 21367.213} C_VEL
LIN {X 0,Y 434.419,Z 678.55,A -85,B 0,C 180,E1 21363.375,E2 21363.375} C_VEL
LIN {X 0,Y 434.411,Z 678.553,A -85,B 0,C 180,E1 21359.535,E2 21359.535} C_VEL
LIN {X 0,Y 434.419,Z 678.554,A -85,B 0,C 180,E1 21355.641,E2 21355.641} C_VEL
LIN {X 0,Y 434.424,Z 678.554,A -85,B 0,C 180,E1 21351.894,E2 21351.894} C_VEL
LIN {X 0,Y 434.421,Z 678.557,A -85,B 0,C 180,E1 21348.086,E2 21348.086} C_VEL
LIN {X 0,Y 434.413,Z 678.548,A -85,B 0,C 180,E1 21344.259,E2 21344.259} C_VEL
LIN {X 0,Y 434.42,Z 678.554,A -85,B 0,C 180,E1 21340.478,E2 21340.478} C_VEL
LIN {X 0,Y 434.411,Z 678.554,A -85,B 0,C 180,E1 21336.61,E2 21336.61} C_VEL
LIN {X 0,Y 434.409,Z 678.551,A -85,B 0,C 180,E1 21332.772,E2 21332.772} C_VEL
LIN {X 0,Y 434.423,Z 678.546,A -85,B 0,C 180,E1 21328.947,E2 21328.947} C_VEL
LIN {X 0,Y 434.421,Z 678.547,A -85,B 0,C 180,E1 21325.117,E2 21325.117} C_VEL
LIN {X 0,Y 434.412,Z 678.552,A -85,B 0,C 180,E1 21321.264,E2 21321.264} C_VEL
LIN {X 0,Y 434.416,Z 678.557,A -85,B 0,C 180,E1 21317.372,E2 21317.372} C_VEL
LIN {X 0,Y 434.411,Z 678.557,A -85,B 0,C 180,E1 21313.694,E2 21313.694} C_VEL
LIN {X 0,Y 434.412,Z 678.55,A -85,B 0,C 180,E1 21309.846,E2 21309.846} C_VEL
LIN {X 0,Y 433.417,Z 678.683,A -85,B 0,C 180,E1 21308.831,E2 21308.831} C_VEL
LIN {X 0,Y 426.916,Z 679.492,A -85,B 0,C 180,E1 21305.895,E2 21305.895} C_VEL
LIN {X 0,Y 426.486,Z 679.538,A -85,B 0,C 180,E1 21305.222,E2 21305.222} C_VEL
LIN {X 0,Y 426.475,Z 679.547,A -85,B 0,C 180,E1 21301.429,E2 21301.429} C_VEL
LIN {X 0,Y 426.487,Z 679.575,A -85,B 0,C 180,E1 21301.022,E2 21301.022} C_VEL
LIN {X 0,Y 427.618,Z 682.747,A -85,B 0,C 180,E1 21300.44,E2 21300.44} C_VEL
LIN {X 0,Y 433.438,Z 695.822,A -85,B 0,C 180,E1 21297.958,E2 21297.958} C_VEL
LIN {X 0,Y 440.567,Z 712.928,A -85,B 0,C 180,E1 21294.959,E2 21294.959} C_VEL
LIN {X 0,Y 447.74,Z 731.603,A -85,B 0,C 180,E1 21291.952,E2 21291.952} C_VEL
LIN {X 0,Y 454.871,Z 752.16,A -85,B 0,C 180,E1 21288.912,E2 21288.912} C_VEL
LIN {X 0,Y 458.437,Z 763.82,A -85,B 0,C 180,E1 21287.31,E2 21287.31} C_VEL
LIN {X 0,Y 453.063,Z 804.028,A -85,B 0,C 180,E1 21283.517,E2 21283.517} C_VEL
LIN {X 0,Y 447.951,Z 845.971,A -85,B 0,C 180,E1 21279.598,E2 21279.598} C_VEL
LIN {X 0,Y 443.177,Z 890.024,A -85,B 0,C 180,E1 21275.511,E2 21275.511} C_VEL
LIN {X 0,Y 440.843,Z 915.013,A -85,B 0,C 180,E1 21273.246,E2 21273.246} C_VEL
LIN {X 0,Y 441.569,Z 927.123,A -85,B 0,C 180,E1 21272.876,E2 21272.876} C_VEL
LIN {X 0,Y 436.419,Z 1024.672,A -85,B 0,C 180,E1 21270.349,E2 21270.349} C_VEL
LIN {X 0,Y 434.742,Z 1065.338,A -85,B 0,C 180,E1 21269.151,E2 21269.151} C_VEL
LIN {X 0,Y 433.914,Z 1082.867,A -85,B 0,C 180,E1 21268.377,E2 21268.377} C_VEL
LIN {X 0,Y 432.843,Z 1099.465,A -85,B 0,C 180,E1 21267.368,E2 21267.368} C_VEL
LIN {X 0,Y 431.65,Z 1114.581,A -85,B 0,C 180,E1 21266.186,E2 21266.186} C_VEL
LIN {X 0,Y 430.383,Z 1129.402,A -85,B 0,C 180,E1 21264.72,E2 21264.72} C_VEL
LIN {X 0,Y 429.21,Z 1141.945,A -85,B 0,C 180,E1 21263.185,E2 21263.185} C_VEL
LIN {X 0,Y 428.064,Z 1153.979,A -85,B 0,C 180,E1 21261.37,E2 21261.37} C_VEL
LIN {X 0,Y 427.161,Z 1163.672,A -85,B 0,C 180,E1 21259.556,E2 21259.556} C_VEL
LIN {X 0,Y 426.409,Z 1172.907,A -85,B 0,C 180,E1 21257.383,E2 21257.383} C_VEL
LIN {X 0,Y 425.943,Z 1179.781,A -85,B 0,C 180,E1 21255.243,E2 21255.243} C_VEL
LIN {X 0,Y 425.737,Z 1184.985,A -85,B 0,C 180,E1 21253.03,E2 21253.03} C_VEL
LIN {X 0,Y 425.761,Z 1188.463,A -85,B 0,C 180,E1 21250.692,E2 21250.692} C_VEL
LIN {X 0,Y 426.026,Z 1190.046,A -85,B 0,C 180,E1 21248.503,E2 21248.503} C_VEL
LIN {X 0,Y 426.557,Z 1189.856,A -85,B 0,C 180,E1 21246.19,E2 21246.19} C_VEL
LIN {X 0,Y 427.377,Z 1188.061,A -85,B 0,C 180,E1 21244.025,E2 21244.025} C_VEL
LIN {X 0,Y 428.622,Z 1184.311,A -85,B 0,C 180,E1 21241.738,E2 21241.738} C_VEL
LIN {X 0,Y 430.203,Z 1179.048,A -85,B 0,C 180,E1 21239.6,E2 21239.6} C_VEL
LIN {X 0,Y 432.356,Z 1171.333,A -85,B 0,C 180,E1 21237.349,E2 21237.349} C_VEL
LIN {X 0,Y 434.679,Z 1162.502,A -85,B 0,C 180,E1 21235.382,E2 21235.382} C_VEL
LIN {X 0,Y 437.205,Z 1152.27,A -85,B 0,C 180,E1 21233.566,E2 21233.566} C_VEL
LIN {X 0,Y 440.062,Z 1139.465,A -85,B 0,C 180,E1 21231.77,E2 21231.77} C_VEL
LIN {X 0,Y 442.786,Z 1125.94,A -85,B 0,C 180,E1 21230.249,E2 21230.249} C_VEL
LIN {X 0,Y 445.278,Z 1112.027,A -85,B 0,C 180,E1 21228.996,E2 21228.996} C_VEL
LIN {X 0,Y 447.654,Z 1096.386,A -85,B 0,C 180,E1 21227.88,E2 21227.88} C_VEL
LIN {X 0,Y 449.718,Z 1079.603,A -85,B 0,C 180,E1 21226.958,E2 21226.958} C_VEL
LIN {X 0,Y 454.157,Z 1045.753,A -85,B 0,C 180,E1 21225.497,E2 21225.497} C_VEL
LIN {X 0,Y 461.955,Z 995.104,A -85,B 0,C 180,E1 21223.613,E2 21223.613} C_VEL
LIN {X 0,Y 468.192,Z 950.727,A -85,B 0,C 180,E1 21222.19,E2 21222.19} C_VEL
LIN {X 0,Y 469.045,Z 943.271,A -85,B 0,C 180,E1 21221.937,E2 21221.937} C_VEL
LIN {X 0,Y 468.87,Z 940.186,A -85,B 0,C 180,E1 21221.731,E2 21221.731} C_VEL
LIN {X 0,Y 479.04,Z 905.804,A -85,B 0,C 180,E1 21217.932,E2 21217.932} C_VEL
LIN {X 0,Y 490.758,Z 873.836,A -85,B 0,C 180,E1 21214.28,E2 21214.28} C_VEL
LIN {X 0,Y 503.712,Z 845.354,A -85,B 0,C 180,E1 21210.9,E2 21210.9} C_VEL
LIN {X 0,Y 512.558,Z 829.007,A -85,B 0,C 180,E1 21208.871,E2 21208.871} C_VEL
LIN {X 0,Y 513.571,Z 826.153,A -85,B 0,C 180,E1 21207.098,E2 21207.098} C_VEL
LIN {X 0,Y 514.703,Z 825.091,A -85,B 0,C 180,E1 21205.363,E2 21205.363} C_VEL
LIN {X 0,Y 501.565,Z 848.372,A -85,B 0,C 180,E1 21202.983,E2 21202.983} C_VEL
LIN {X 0,Y 492.599,Z 868.734,A -85,B 0,C 180,E1 21200.745,E2 21200.745} C_VEL
LIN {X 0,Y 486.389,Z 888.583,A -85,B 0,C 180,E1 21198.394,E2 21198.394} C_VEL
LIN {X 0,Y 483.453,Z 905.101,A -85,B 0,C 180,E1 21196.307,E2 21196.307} C_VEL
LIN {X 0,Y 482.795,Z 922.729,A -85,B 0,C 180,E1 21193.971,E2 21193.971} C_VEL
LIN {X 0,Y 484.683,Z 938.625,A -85,B 0,C 180,E1 21191.782,E2 21191.782} C_VEL
LIN {X 0,Y 487.348,Z 949.934,A -85,B 0,C 180,E1 21190.221,E2 21190.221} C_VEL
LIN {X 0,Y 476.502,Z 971.68,A -85,B 0,C 180,E1 21189.322,E2 21189.322} C_VEL
LIN {X 0,Y 467.972,Z 991.759,A -85,B 0,C 180,E1 21188.345,E2 21188.345} C_VEL
LIN {X 0,Y 463.256,Z 1026.863,A -85,B 0,C 180,E1 21187.803,E2 21187.803} C_VEL
LIN {X 0,Y 460.502,Z 1050.778,A -85,B 0,C 180,E1 21187.147,E2 21187.147} C_VEL
LIN {X 0,Y 457.079,Z 1074.876,A -85,B 0,C 180,E1 21186.267,E2 21186.267} C_VEL
LIN {X 0,Y 453.39,Z 1097.45,A -85,B 0,C 180,E1 21185.216,E2 21185.216} C_VEL
LIN {X 0,Y 449.369,Z 1120.35,A -85,B 0,C 180,E1 21183.88,E2 21183.88} C_VEL
LIN {X 0,Y 445.44,Z 1141.707,A -85,B 0,C 180,E1 21182.366,E2 21182.366} C_VEL
LIN {X 0,Y 441.429,Z 1162.8,A -85,B 0,C 180,E1 21180.563,E2 21180.563} C_VEL
LIN {X 0,Y 437.777,Z 1182.076,A -85,B 0,C 180,E1 21178.616,E2 21178.616} C_VEL
LIN {X 0,Y 433.535,Z 1207.911,A -85,B 0,C 180,E1 21175.694,E2 21175.694} C_VEL
LIN {X 0,Y 431.011,Z 1224.22,A -85,B 0,C 180,E1 21173.514,E2 21173.514} C_VEL
LIN {X 0,Y 428.826,Z 1239.149,A -85,B 0,C 180,E1 21171.143,E2 21171.143} C_VEL
LIN {X 0,Y 427.163,Z 1251.42,A -85,B 0,C 180,E1 21168.844,E2 21168.844} C_VEL
LIN {X 0,Y 425.861,Z 1262.68,A -85,B 0,C 180,E1 21166.363,E2 21166.363} C_VEL
LIN {X 0,Y 424.944,Z 1272.537,A -85,B 0,C 180,E1 21163.746,E2 21163.746} C_VEL
LIN {X 0,Y 424.423,Z 1280.449,A -85,B 0,C 180,E1 21161.137,E2 21161.137} C_VEL
LIN {X 0,Y 424.218,Z 1286.99,A -85,B 0,C 180,E1 21158.401,E2 21158.401} C_VEL
LIN {X 0,Y 424.196,Z 1291.43,A -85,B 0,C 180,E1 21155.89,E2 21155.89} C_VEL
LIN {X 0,Y 424.25,Z 1294.513,A -85,B 0,C 180,E1 21153.241,E2 21153.241} C_VEL
LIN {X 0,Y 424.28,Z 1296.072,A -85,B 0,C 180,E1 21150.673,E2 21150.673} C_VEL
LIN {X 0,Y 424.248,Z 1296.039,A -85,B 0,C 180,E1 21148.107,E2 21148.107} C_VEL
LIN {X 0,Y 424.166,Z 1294.667,A -85,B 0,C 180,E1 21145.537,E2 21145.537} C_VEL
LIN {X 0,Y 424.142,Z 1291.521,A -85,B 0,C 180,E1 21142.821,E2 21142.821} C_VEL
LIN {X 0,Y 424.292,Z 1286.531,A -85,B 0,C 180,E1 21139.955,E2 21139.955} C_VEL
LIN {X 0,Y 424.784,Z 1280.102,A -85,B 0,C 180,E1 21137.215,E2 21137.215} C_VEL
LIN {X 0,Y 425.723,Z 1271.779,A -85,B 0,C 180,E1 21134.468,E2 21134.468} C_VEL
LIN {X 0,Y 427.242,Z 1261.606,A -85,B 0,C 180,E1 21131.722,E2 21131.722} C_VEL
LIN {X 0,Y 429.303,Z 1250.08,A -85,B 0,C 180,E1 21129.122,E2 21129.122} C_VEL
LIN {X 0,Y 432.023,Z 1236.381,A -85,B 0,C 180,E1 21126.54,E2 21126.54} C_VEL
LIN {X 0,Y 435.29,Z 1221.177,A -85,B 0,C 180,E1 21124.121,E2 21124.121} C_VEL
LIN {X 0,Y 439.249,Z 1203.556,A -85,B 0,C 180,E1 21121.738,E2 21121.738} C_VEL
LIN {X 0,Y 443.72,Z 1184.212,A -85,B 0,C 180,E1 21119.533,E2 21119.533} C_VEL
LIN {X 0,Y 448.454,Z 1163.802,A -85,B 0,C 180,E1 21117.571,E2 21117.571} C_VEL
LIN {X 0,Y 453.353,Z 1142.575,A -85,B 0,C 180,E1 21115.852,E2 21115.852} C_VEL
LIN {X 0,Y 458.524,Z 1119.757,A -85,B 0,C 180,E1 21114.314,E2 21114.314} C_VEL
LIN {X 0,Y 463.68,Z 1096.182,A -85,B 0,C 180,E1 21113.011,E2 21113.011} C_VEL
LIN {X 0,Y 468.862,Z 1071.138,A -85,B 0,C 180,E1 21111.912,E2 21111.912} C_VEL
LIN {X 0,Y 473.985,Z 1043.301,A -85,B 0,C 180,E1 21110.966,E2 21110.966} C_VEL
LIN {X 0,Y 477.677,Z 1021.511,A -85,B 0,C 180,E1 21110.411,E2 21110.411} C_VEL
LIN {X 0,Y 483.398,Z 992.963,A -85,B 0,C 180,E1 21109.908,E2 21109.908} C_VEL
LIN {X 0,Y 489.264,Z 966.362,A -85,B 0,C 180,E1 21109.552,E2 21109.552} C_VEL
LIN {X 0,Y 493.147,Z 950.075,A -85,B 0,C 180,E1 21109.412,E2 21109.412} C_VEL
LIN {X 0,Y 491.772,Z 938.794,A -85,B 0,C 180,E1 21107.875,E2 21107.875} C_VEL
LIN {X 0,Y 492.125,Z 927.303,A -85,B 0,C 180,E1 21106.329,E2 21106.329} C_VEL
LIN {X 0,Y 493.719,Z 917.64,A -85,B 0,C 180,E1 21105.085,E2 21105.085} C_VEL
LIN {X 0,Y 497.1,Z 905.847,A -85,B 0,C 180,E1 21103.582,E2 21103.582} C_VEL
LIN {X 0,Y 500.743,Z 896.434,A -85,B 0,C 180,E1 21102.517,E2 21102.517} C_VEL
LIN {X 0,Y 486.913,Z 963.995,A -85,B 0,C 180,E1 21100.62,E2 21100.62} C_VEL
LIN {X 0,Y 475.491,Z 1031.306,A -85,B 0,C 180,E1 21098.678,E2 21098.678} C_VEL
LIN {X 0,Y 471.243,Z 1054.897,A -85,B 0,C 180,E1 21097.745,E2 21097.745} C_VEL
LIN {X 0,Y 466.542,Z 1078.321,A -85,B 0,C 180,E1 21096.571,E2 21096.571} C_VEL
LIN {X 0,Y 461.643,Z 1100.814,A -85,B 0,C 180,E1 21095.18,E2 21095.18} C_VEL
LIN {X 0,Y 456.647,Z 1122.365,A -85,B 0,C 180,E1 21093.565,E2 21093.565} C_VEL
LIN {X 0,Y 451.656,Z 1142.845,A -85,B 0,C 180,E1 21091.721,E2 21091.721} C_VEL
LIN {X 0,Y 446.888,Z 1161.587,A -85,B 0,C 180,E1 21089.709,E2 21089.709} C_VEL
LIN {X 0,Y 442.788,Z 1177.264,A -85,B 0,C 180,E1 21087.722,E2 21087.722} C_VEL
LIN {X 0,Y 438.637,Z 1193.009,A -85,B 0,C 180,E1 21085.376,E2 21085.376} C_VEL
LIN {X 0,Y 435.116,Z 1206.496,A -85,B 0,C 180,E1 21082.996,E2 21082.996} C_VEL
LIN {X 0,Y 432.037,Z 1218.608,A -85,B 0,C 180,E1 21080.455,E2 21080.455} C_VEL
LIN {X 0,Y 429.445,Z 1229.173,A -85,B 0,C 180,E1 21077.759,E2 21077.759} C_VEL
LIN {X 0,Y 427.481,Z 1237.835,A -85,B 0,C 180,E1 21075.048,E2 21075.048} C_VEL
LIN {X 0,Y 426.025,Z 1245.082,A -85,B 0,C 180,E1 21072.195,E2 21072.195} C_VEL
LIN {X 0,Y 425.08,Z 1250.566,A -85,B 0,C 180,E1 21069.341,E2 21069.341} C_VEL
LIN {X 0,Y 424.538,Z 1254.241,A -85,B 0,C 180,E1 21066.491,E2 21066.491} C_VEL
LIN {X 0,Y 424.253,Z 1256.298,A -85,B 0,C 180,E1 21063.648,E2 21063.648} C_VEL
LIN {X 0,Y 424.15,Z 1256.805,A -85,B 0,C 180,E1 21060.946,E2 21060.946} C_VEL
LIN {X 0,Y 424.112,Z 1255.699,A -85,B 0,C 180,E1 21058.244,E2 21058.244} C_VEL
LIN {X 0,Y 424.153,Z 1252.966,A -85,B 0,C 180,E1 21055.403,E2 21055.403} C_VEL
LIN {X 0,Y 424.339,Z 1248.823,A -85,B 0,C 180,E1 21052.69,E2 21052.69} C_VEL
LIN {X 0,Y 424.717,Z 1242.925,A -85,B 0,C 180,E1 21049.967,E2 21049.967} C_VEL
LIN {X 0,Y 425.413,Z 1235.311,A -85,B 0,C 180,E1 21047.236,E2 21047.236} C_VEL
LIN {X 0,Y 426.441,Z 1226.356,A -85,B 0,C 180,E1 21044.636,E2 21044.636} C_VEL
LIN {X 0,Y 427.943,Z 1215.21,A -85,B 0,C 180,E1 21041.984,E2 21041.984} C_VEL
LIN {X 0,Y 429.747,Z 1203.042,A -85,B 0,C 180,E1 21039.573,E2 21039.573} C_VEL
LIN {X 0,Y 432.067,Z 1188.417,A -85,B 0,C 180,E1 21037.121,E2 21037.121} C_VEL
LIN {X 0,Y 434.654,Z 1172.659,A -85,B 0,C 180,E1 21034.885,E2 21034.885} C_VEL
LIN {X 0,Y 437.369,Z 1156.076,A -85,B 0,C 180,E1 21032.879,E2 21032.879} C_VEL
LIN {X 0,Y 440.304,Z 1137.55,A -85,B 0,C 180,E1 21030.99,E2 21030.99} C_VEL
LIN {X 0,Y 443.165,Z 1118.408,A -85,B 0,C 180,E1 21029.342,E2 21029.342} C_VEL
LIN {X 0,Y 446.074,Z 1097.51,A -85,B 0,C 180,E1 21027.834,E2 21027.834} C_VEL
LIN {X 0,Y 448.66,Z 1076.836,A -85,B 0,C 180,E1 21026.601,E2 21026.601} C_VEL
LIN {X 0,Y 451.043,Z 1054.981,A -85,B 0,C 180,E1 21025.542,E2 21025.542} C_VEL
LIN {X 0,Y 453.148,Z 1031.49,A -85,B 0,C 180,E1 21024.667,E2 21024.667} C_VEL
LIN {X 0,Y 454.71,Z 1008.646,A -85,B 0,C 180,E1 21024.047,E2 21024.047} C_VEL
LIN {X 0,Y 467.989,Z 766.151,A -85,B 0,C 180,E1 21019.194,E2 21019.194} C_VEL
LIN {X 0,Y 452.016,Z 734.877,A -85,B 0,C 180,E1 21017.002,E2 21017.002} C_VEL
LIN {X 0,Y 438.049,Z 709.106,A -85,B 0,C 180,E1 21014.959,E2 21014.959} C_VEL
LIN {X 0,Y 430.627,Z 690.024,A -85,B 0,C 180,E1 21011.97,E2 21011.97} C_VEL
LIN {X 0,Y 426.475,Z 679.54,A -85,B 0,C 180,E1 21010.228,E2 21010.228} C_VEL
LIN {X 0,Y 426.481,Z 679.54,A -85,B 0,C 180,E1 21006.383,E2 21006.383} C_VEL
LIN {X 0,Y 426.487,Z 679.546,A -85,B 0,C 180,E1 21002.433,E2 21002.433} C_VEL
LIN {X 0,Y 426.475,Z 679.543,A -85,B 0,C 180,E1 20998.575,E2 20998.575} C_VEL
LIN {X 0,Y 426.476,Z 679.544,A -85,B 0,C 180,E1 20994.668,E2 20994.668} C_VEL
LIN {X 0,Y 426.483,Z 679.543,A -85,B 0,C 180,E1 20990.879,E2 20990.879} C_VEL
LIN {X 0,Y 426.473,Z 679.543,A -85,B 0,C 180,E1 20987.043,E2 20987.043} C_VEL
LIN {X 0,Y 426.478,Z 679.53,A -85,B 0,C 180,E1 20983.147,E2 20983.147} C_VEL
LIN {X 0,Y 426.474,Z 679.534,A -85,B 0,C 180,E1 20979.312,E2 20979.312} C_VEL
LIN {X 0,Y 426.477,Z 679.542,A -85,B 0,C 180,E1 20975.518,E2 20975.518} C_VEL
LIN {X 0,Y 426.471,Z 679.544,A -85,B 0,C 180,E1 20971.614,E2 20971.614} C_VEL
LIN {X 0,Y 426.478,Z 679.544,A -85,B 0,C 180,E1 20967.852,E2 20967.852} C_VEL
LIN {X 0,Y 426.478,Z 679.545,A -85,B 0,C 180,E1 20963.946,E2 20963.946} C_VEL
LIN {X 0,Y 426.473,Z 679.547,A -85,B 0,C 180,E1 20960.147,E2 20960.147} C_VEL
LIN {X 0,Y 426.487,Z 679.539,A -85,B 0,C 180,E1 20956.305,E2 20956.305} C_VEL
LIN {X 0,Y 426.483,Z 679.539,A -85,B 0,C 180,E1 20952.398,E2 20952.398} C_VEL
LIN {X 0,Y 426.475,Z 679.548,A -85,B 0,C 180,E1 20948.549,E2 20948.549} C_VEL
LIN {X 0,Y 426.486,Z 679.538,A -85,B 0,C 180,E1 20945.222,E2 20945.222} C_VEL
LIN {X 0,Y 425.482,Z 679.665,A -85,B 0,C 180,E1 20944.534,E2 20944.534} C_VEL
LIN {X 0,Y 419.078,Z 680.462,A -85,B 0,C 180,E1 20942.662,E2 20942.662} C_VEL
LIN {X 0,Y 418.544,Z 680.529,A -85,B 0,C 180,E1 20942.153,E2 20942.153} C_VEL
LIN {X 0,Y 418.582,Z 680.777,A -85,B 0,C 180,E1 20942.008,E2 20942.008} C_VEL
LIN {X 0,Y 419.784,Z 683.931,A -85,B 0,C 180,E1 20941.398,E2 20941.398} C_VEL
LIN {X 0,Y 425.286,Z 696.028,A -85,B 0,C 180,E1 20939.013,E2 20939.013} C_VEL
LIN {X 0,Y 432.929,Z 714.382,A -85,B 0,C 180,E1 20935.702,E2 20935.702} C_VEL
LIN {X 0,Y 440.055,Z 732.807,A -85,B 0,C 180,E1 20932.653,E2 20932.653} C_VEL
LIN {X 0,Y 447,Z 752.607,A -85,B 0,C 180,E1 20929.644,E2 20929.644} C_VEL
LIN {X 0,Y 451.379,Z 766.515,A -85,B 0,C 180,E1 20927.672,E2 20927.672} C_VEL
LIN {X 0,Y 445.77,Z 807.249,A -85,B 0,C 180,E1 20923.792,E2 20923.792} C_VEL
LIN {X 0,Y 440.39,Z 850.166,A -85,B 0,C 180,E1 20919.737,E2 20919.737} C_VEL
LIN {X 0,Y 435.396,Z 895.094,A -85,B 0,C 180,E1 20915.522,E2 20915.522} C_VEL
LIN {X 0,Y 433.431,Z 915.754,A -85,B 0,C 180,E1 20913.634,E2 20913.634} C_VEL
LIN {X 0,Y 434.136,Z 927.8,A -85,B 0,C 180,E1 20913.259,E2 20913.259} C_VEL
LIN {X 0,Y 429.054,Z 1019.954,A -85,B 0,C 180,E1 20910.805,E2 20910.805} C_VEL
LIN {X 0,Y 427.047,Z 1065.432,A -85,B 0,C 180,E1 20909.444,E2 20909.444} C_VEL
LIN {X 0,Y 426.215,Z 1082.663,A -85,B 0,C 180,E1 20908.676,E2 20908.676} C_VEL
LIN {X 0,Y 425.143,Z 1099.089,A -85,B 0,C 180,E1 20907.678,E2 20907.678} C_VEL
LIN {X 0,Y 423.911,Z 1114.448,A -85,B 0,C 180,E1 20906.475,E2 20906.475} C_VEL
LIN {X 0,Y 422.637,Z 1128.991,A -85,B 0,C 180,E1 20905.032,E2 20905.032} C_VEL
LIN {X 0,Y 421.385,Z 1142.172,A -85,B 0,C 180,E1 20903.419,E2 20903.419} C_VEL
LIN {X 0,Y 420.152,Z 1154.781,A -85,B 0,C 180,E1 20901.493,E2 20901.493} C_VEL
LIN {X 0,Y 419.201,Z 1164.738,A -85,B 0,C 180,E1 20899.59,E2 20899.59} C_VEL
LIN {X 0,Y 418.439,Z 1173.92,A -85,B 0,C 180,E1 20897.379,E2 20897.379} C_VEL
LIN {X 0,Y 417.96,Z 1181.01,A -85,B 0,C 180,E1 20895.115,E2 20895.115} C_VEL
LIN {X 0,Y 417.772,Z 1186.146,A -85,B 0,C 180,E1 20892.861,E2 20892.861} C_VEL
LIN {X 0,Y 417.832,Z 1189.651,A -85,B 0,C 180,E1 20890.425,E2 20890.425} C_VEL
LIN {X 0,Y 418.152,Z 1191.133,A -85,B 0,C 180,E1 20888.11,E2 20888.11} C_VEL
LIN {X 0,Y 418.779,Z 1190.841,A -85,B 0,C 180,E1 20885.755,E2 20885.755} C_VEL
LIN {X 0,Y 419.764,Z 1188.704,A -85,B 0,C 180,E1 20883.414,E2 20883.414} C_VEL
LIN {X 0,Y 421.175,Z 1184.765,A -85,B 0,C 180,E1 20881.088,E2 20881.088} C_VEL
LIN {X 0,Y 423.054,Z 1178.795,A -85,B 0,C 180,E1 20878.781,E2 20878.781} C_VEL
LIN {X 0,Y 425.159,Z 1171.805,A -85,B 0,C 180,E1 20876.764,E2 20876.764} C_VEL
LIN {X 0,Y 427.846,Z 1162.192,A -85,B 0,C 180,E1 20874.636,E2 20874.636} C_VEL
LIN {X 0,Y 430.777,Z 1150.752,A -85,B 0,C 180,E1 20872.665,E2 20872.665} C_VEL
LIN {X 0,Y 433.545,Z 1139.045,A -85,B 0,C 180,E1 20871.044,E2 20871.044} C_VEL
LIN {X 0,Y 436.335,Z 1125.899,A -85,B 0,C 180,E1 20869.57,E2 20869.57} C_VEL
LIN {X 0,Y 439.413,Z 1109.483,A -85,B 0,C 180,E1 20868.116,E2 20868.116} C_VEL
LIN {X 0,Y 441.955,Z 1093.055,A -85,B 0,C 180,E1 20866.991,E2 20866.991} C_VEL
LIN {X 0,Y 444.518,Z 1072.608,A -85,B 0,C 180,E1 20865.94,E2 20865.94} C_VEL
LIN {X 0,Y 450.014,Z 1036.794,A -85,B 0,C 180,E1 20864.404,E2 20864.404} C_VEL
LIN {X 0,Y 457.864,Z 988.463,A -85,B 0,C 180,E1 20862.608,E2 20862.608} C_VEL
LIN {X 0,Y 463.931,Z 945.403,A -85,B 0,C 180,E1 20861.215,E2 20861.215} C_VEL
LIN {X 0,Y 463.791,Z 941.465,A -85,B 0,C 180,E1 20860.936,E2 20860.936} C_VEL
LIN {X 0,Y 474.713,Z 907.037,A -85,B 0,C 180,E1 20857.066,E2 20857.066} C_VEL
LIN {X 0,Y 487.451,Z 874.724,A -85,B 0,C 180,E1 20853.306,E2 20853.306} C_VEL
LIN {X 0,Y 501.14,Z 846.899,A -85,B 0,C 180,E1 20849.947,E2 20849.947} C_VEL
LIN {X 0,Y 508.122,Z 834.81,A -85,B 0,C 180,E1 20848.432,E2 20848.432} C_VEL
LIN {X 0,Y 509.123,Z 832.53,A -85,B 0,C 180,E1 20846.774,E2 20846.774} C_VEL
LIN {X 0,Y 509.766,Z 831.957,A -85,B 0,C 180,E1 20845.763,E2 20845.763} C_VEL
LIN {X 0,Y 496.667,Z 854.481,A -85,B 0,C 180,E1 20843.422,E2 20843.422} C_VEL
LIN {X 0,Y 487.576,Z 874.264,A -85,B 0,C 180,E1 20841.191,E2 20841.191} C_VEL
LIN {X 0,Y 481.383,Z 892.868,A -85,B 0,C 180,E1 20838.934,E2 20838.934} C_VEL
LIN {X 0,Y 477.976,Z 910.329,A -85,B 0,C 180,E1 20836.673,E2 20836.673} C_VEL
LIN {X 0,Y 477.082,Z 927.145,A -85,B 0,C 180,E1 20834.382,E2 20834.382} C_VEL
LIN {X 0,Y 478.776,Z 943.35,A -85,B 0,C 180,E1 20832.094,E2 20832.094} C_VEL
LIN {X 0,Y 480.687,Z 952.178,A -85,B 0,C 180,E1 20830.836,E2 20830.836} C_VEL
LIN {X 0,Y 469.85,Z 974.078,A -85,B 0,C 180,E1 20829.91,E2 20829.91} C_VEL
LIN {X 0,Y 462.819,Z 990.592,A -85,B 0,C 180,E1 20829.1,E2 20829.1} C_VEL
LIN {X 0,Y 457.784,Z 1026.768,A -85,B 0,C 180,E1 20828.531,E2 20828.531} C_VEL
LIN {X 0,Y 454.821,Z 1050.382,A -85,B 0,C 180,E1 20827.863,E2 20827.863} C_VEL
LIN {X 0,Y 451.027,Z 1075.496,A -85,B 0,C 180,E1 20826.923,E2 20826.923} C_VEL
LIN {X 0,Y 447.162,Z 1097.653,A -85,B 0,C 180,E1 20825.86,E2 20825.86} C_VEL
LIN {X 0,Y 442.768,Z 1121.285,A -85,B 0,C 180,E1 20824.448,E2 20824.448} C_VEL
LIN {X 0,Y 438.511,Z 1142.829,A -85,B 0,C 180,E1 20822.864,E2 20822.864} C_VEL
LIN {X 0,Y 434.208,Z 1164.328,A -85,B 0,C 180,E1 20820.973,E2 20820.973} C_VEL
LIN {X 0,Y 430.108,Z 1184.492,A -85,B 0,C 180,E1 20818.839,E2 20818.839} C_VEL
LIN {X 0,Y 424.268,Z 1217.109,A -85,B 0,C 180,E1 20814.726,E2 20814.726} C_VEL
LIN {X 0,Y 421.888,Z 1232.491,A -85,B 0,C 180,E1 20812.429,E2 20812.429} C_VEL
LIN {X 0,Y 419.938,Z 1245.911,A -85,B 0,C 180,E1 20810.05,E2 20810.05} C_VEL
LIN {X 0,Y 418.393,Z 1257.959,A -85,B 0,C 180,E1 20807.523,E2 20807.523} C_VEL
LIN {X 0,Y 417.272,Z 1268.601,A -85,B 0,C 180,E1 20804.854,E2 20804.854} C_VEL
LIN {X 0,Y 416.6,Z 1277.317,A -85,B 0,C 180,E1 20802.191,E2 20802.191} C_VEL
LIN {X 0,Y 416.279,Z 1284.143,A -85,B 0,C 180,E1 20799.538,E2 20799.538} C_VEL
LIN {X 0,Y 416.201,Z 1289.616,A -85,B 0,C 180,E1 20796.758,E2 20796.758} C_VEL
LIN {X 0,Y 416.24,Z 1293.036,A -85,B 0,C 180,E1 20794.269,E2 20794.269} C_VEL
LIN {X 0,Y 416.294,Z 1295.219,A -85,B 0,C 180,E1 20791.512,E2 20791.512} C_VEL
LIN {X 0,Y 416.277,Z 1295.823,A -85,B 0,C 180,E1 20788.897,E2 20788.897} C_VEL
LIN {X 0,Y 416.194,Z 1294.859,A -85,B 0,C 180,E1 20786.279,E2 20786.279} C_VEL
LIN {X 0,Y 416.126,Z 1292.381,A -85,B 0,C 180,E1 20783.514,E2 20783.514} C_VEL
LIN {X 0,Y 416.217,Z 1288.177,A -85,B 0,C 180,E1 20780.736,E2 20780.736} C_VEL
LIN {X 0,Y 416.642,Z 1282.032,A -85,B 0,C 180,E1 20777.806,E2 20777.806} C_VEL
LIN {X 0,Y 417.508,Z 1274.458,A -85,B 0,C 180,E1 20775.008,E2 20775.008} C_VEL
LIN {X 0,Y 418.952,Z 1264.937,A -85,B 0,C 180,E1 20772.211,E2 20772.211} C_VEL
LIN {X 0,Y 421.061,Z 1253.445,A -85,B 0,C 180,E1 20769.422,E2 20769.422} C_VEL
LIN {X 0,Y 423.767,Z 1240.539,A -85,B 0,C 180,E1 20766.792,E2 20766.792} C_VEL
LIN {X 0,Y 427.036,Z 1226.273,A -85,B 0,C 180,E1 20764.329,E2 20764.329} C_VEL
LIN {X 0,Y 431.007,Z 1209.63,A -85,B 0,C 180,E1 20761.903,E2 20761.903} C_VEL
LIN {X 0,Y 435.358,Z 1191.984,A -85,B 0,C 180,E1 20759.719,E2 20759.719} C_VEL
LIN {X 0,Y 440.393,Z 1171.824,A -85,B 0,C 180,E1 20757.599,E2 20757.599} C_VEL
LIN {X 0,Y 445.889,Z 1149.9,A -85,B 0,C 180,E1 20755.667,E2 20755.667} C_VEL
LIN {X 0,Y 451.551,Z 1127,A -85,B 0,C 180,E1 20753.99,E2 20753.99} C_VEL
LIN {X 0,Y 457.266,Z 1103.247,A -85,B 0,C 180,E1 20752.561,E2 20752.561} C_VEL
LIN {X 0,Y 462.681,Z 1079.874,A -85,B 0,C 180,E1 20751.429,E2 20751.429} C_VEL
LIN {X 0,Y 468.284,Z 1053.568,A -85,B 0,C 180,E1 20750.427,E2 20750.427} C_VEL
LIN {X 0,Y 473.127,Z 1027.866,A -85,B 0,C 180,E1 20749.671,E2 20749.671} C_VEL
LIN {X 0,Y 479.412,Z 997.219,A -85,B 0,C 180,E1 20749.087,E2 20749.087} C_VEL
LIN {X 0,Y 486.4,Z 966.584,A -85,B 0,C 180,E1 20748.674,E2 20748.674} C_VEL
LIN {X 0,Y 489.596,Z 953.31,A -85,B 0,C 180,E1 20748.549,E2 20748.549} C_VEL
LIN {X 0,Y 489.196,Z 939.734,A -85,B 0,C 180,E1 20746.624,E2 20746.624} C_VEL
LIN {X 0,Y 491.013,Z 927.87,A -85,B 0,C 180,E1 20745.079,E2 20745.079} C_VEL
LIN {X 0,Y 494.827,Z 915.114,A -85,B 0,C 180,E1 20743.373,E2 20743.373} C_VEL
LIN {X 0,Y 495.931,Z 912.332,A -85,B 0,C 180,E1 20743,E2 20743} C_VEL
LIN {X 0,Y 481.627,Z 978.928,A -85,B 0,C 180,E1 20741.112,E2 20741.112} C_VEL
LIN {X 0,Y 471.74,Z 1032.777,A -85,B 0,C 180,E1 20739.515,E2 20739.515} C_VEL
LIN {X 0,Y 466.977,Z 1056.691,A -85,B 0,C 180,E1 20738.542,E2 20738.542} C_VEL
LIN {X 0,Y 461.754,Z 1080.294,A -85,B 0,C 180,E1 20737.324,E2 20737.324} C_VEL
LIN {X 0,Y 456.353,Z 1102.932,A -85,B 0,C 180,E1 20735.881,E2 20735.881} C_VEL
LIN {X 0,Y 450.858,Z 1124.659,A -85,B 0,C 180,E1 20734.201,E2 20734.201} C_VEL
LIN {X 0,Y 445.435,Z 1145.162,A -85,B 0,C 180,E1 20732.293,E2 20732.293} C_VEL
LIN {X 0,Y 440.27,Z 1164.015,A -85,B 0,C 180,E1 20730.202,E2 20730.202} C_VEL
LIN {X 0,Y 435.446,Z 1181.203,A -85,B 0,C 180,E1 20727.933,E2 20727.933} C_VEL
LIN {X 0,Y 431.147,Z 1196.323,A -85,B 0,C 180,E1 20725.554,E2 20725.554} C_VEL
LIN {X 0,Y 427.481,Z 1209.278,A -85,B 0,C 180,E1 20723.139,E2 20723.139} C_VEL
LIN {X 0,Y 424.13,Z 1221.489,A -85,B 0,C 180,E1 20720.421,E2 20720.421} C_VEL
LIN {X 0,Y 421.615,Z 1231.223,A -85,B 0,C 180,E1 20717.814,E2 20717.814} C_VEL
LIN {X 0,Y 419.499,Z 1239.961,A -85,B 0,C 180,E1 20714.917,E2 20714.917} C_VEL
LIN {X 0,Y 418.018,Z 1246.766,A -85,B 0,C 180,E1 20712.011,E2 20712.011} C_VEL
LIN {X 0,Y 417.032,Z 1252.029,A -85,B 0,C 180,E1 20708.966,E2 20708.966} C_VEL
LIN {X 0,Y 416.51,Z 1255.366,A -85,B 0,C 180,E1 20706.063,E2 20706.063} C_VEL
LIN {X 0,Y 416.247,Z 1256.969,A -85,B 0,C 180,E1 20703.305,E2 20703.305} C_VEL
LIN {X 0,Y 416.144,Z 1257.045,A -85,B 0,C 180,E1 20700.413,E2 20700.413} C_VEL
LIN {X 0,Y 416.119,Z 1255.649,A -85,B 0,C 180,E1 20697.659,E2 20697.659} C_VEL
LIN {X 0,Y 416.182,Z 1252.636,A -85,B 0,C 180,E1 20694.9,E2 20694.9} C_VEL
LIN {X 0,Y 416.41,Z 1247.799,A -85,B 0,C 180,E1 20691.994,E2 20691.994} C_VEL
LIN {X 0,Y 416.87,Z 1241.526,A -85,B 0,C 180,E1 20689.217,E2 20689.217} C_VEL
LIN {X 0,Y 417.641,Z 1233.845,A -85,B 0,C 180,E1 20686.571,E2 20686.571} C_VEL
LIN {X 0,Y 418.797,Z 1224.377,A -85,B 0,C 180,E1 20683.921,E2 20683.921} C_VEL
LIN {X 0,Y 420.414,Z 1212.974,A -85,B 0,C 180,E1 20681.272,E2 20681.272} C_VEL
LIN {X 0,Y 422.428,Z 1200.131,A -85,B 0,C 180,E1 20678.767,E2 20678.767} C_VEL
LIN {X 0,Y 424.789,Z 1185.742,A -85,B 0,C 180,E1 20676.412,E2 20676.412} C_VEL
LIN {X 0,Y 427.437,Z 1169.907,A -85,B 0,C 180,E1 20674.208,E2 20674.208} C_VEL
LIN {X 0,Y 430.438,Z 1151.971,A -85,B 0,C 180,E1 20672.09,E2 20672.09} C_VEL
LIN {X 0,Y 433.383,Z 1133.687,A -85,B 0,C 180,E1 20670.261,E2 20670.261} C_VEL
LIN {X 0,Y 436.42,Z 1113.823,A -85,B 0,C 180,E1 20668.585,E2 20668.585} C_VEL
LIN {X 0,Y 439.335,Z 1092.91,A -85,B 0,C 180,E1 20667.122,E2 20667.122} C_VEL
LIN {X 0,Y 441.974,Z 1071.512,A -85,B 0,C 180,E1 20665.897,E2 20665.897} C_VEL
LIN {X 0,Y 444.365,Z 1049.086,A -85,B 0,C 180,E1 20664.867,E2 20664.867} C_VEL
LIN {X 0,Y 446.375,Z 1025.796,A -85,B 0,C 180,E1 20664.044,E2 20664.044} C_VEL
LIN {X 0,Y 447.957,Z 1002.051,A -85,B 0,C 180,E1 20663.441,E2 20663.441} C_VEL
LIN {X 0,Y 461.063,Z 772.877,A -85,B 0,C 180,E1 20658.78,E2 20658.78} C_VEL
LIN {X 0,Y 461.18,Z 768.686,A -85,B 0,C 180,E1 20658.684,E2 20658.684} C_VEL
LIN {X 0,Y 444.45,Z 735.94,A -85,B 0,C 180,E1 20656.328,E2 20656.328} C_VEL
LIN {X 0,Y 429.948,Z 709.409,A -85,B 0,C 180,E1 20654.15,E2 20654.15} C_VEL
LIN {X 0,Y 422.529,Z 690.659,A -85,B 0,C 180,E1 20651.139,E2 20651.139} C_VEL
LIN {X 0,Y 418.545,Z 680.529,A -85,B 0,C 180,E1 20649.456,E2 20649.456} C_VEL
LIN {X 0,Y 418.545,Z 680.536,A -85,B 0,C 180,E1 20645.657,E2 20645.657} C_VEL
LIN {X 0,Y 418.533,Z 680.529,A -85,B 0,C 180,E1 20641.709,E2 20641.709} C_VEL
LIN {X 0,Y 418.54,Z 680.53,A -85,B 0,C 180,E1 20637.88,E2 20637.88} C_VEL
LIN {X 0,Y 418.543,Z 680.532,A -85,B 0,C 180,E1 20633.963,E2 20633.963} C_VEL
LIN {X 0,Y 418.548,Z 680.533,A -85,B 0,C 180,E1 20630.123,E2 20630.123} C_VEL
LIN {X 0,Y 418.533,Z 680.533,A -85,B 0,C 180,E1 20626.233,E2 20626.233} C_VEL
LIN {X 0,Y 418.542,Z 680.521,A -85,B 0,C 180,E1 20622.418,E2 20622.418} C_VEL
LIN {X 0,Y 418.535,Z 680.517,A -85,B 0,C 180,E1 20618.52,E2 20618.52} C_VEL
LIN {X 0,Y 418.531,Z 680.525,A -85,B 0,C 180,E1 20614.661,E2 20614.661} C_VEL
LIN {X 0,Y 418.54,Z 680.526,A -85,B 0,C 180,E1 20610.686,E2 20610.686} C_VEL
LIN {X 0,Y 418.535,Z 680.527,A -85,B 0,C 180,E1 20606.852,E2 20606.852} C_VEL
LIN {X 0,Y 418.537,Z 680.526,A -85,B 0,C 180,E1 20603.004,E2 20603.004} C_VEL
LIN {X 0,Y 418.53,Z 680.523,A -85,B 0,C 180,E1 20599.084,E2 20599.084} C_VEL
LIN {X 0,Y 418.539,Z 680.527,A -85,B 0,C 180,E1 20595.192,E2 20595.192} C_VEL
LIN {X 0,Y 418.543,Z 680.536,A -85,B 0,C 180,E1 20591.332,E2 20591.332} C_VEL
LIN {X 0,Y 418.537,Z 680.528,A -85,B 0,C 180,E1 20587.382,E2 20587.382} C_VEL
LIN {X 0,Y 418.545,Z 680.532,A -85,B 0,C 180,E1 20583.468,E2 20583.468} C_VEL
LIN {X 0,Y 418.544,Z 680.529,A -85,B 0,C 180,E1 20582.153,E2 20582.153} C_VEL
LIN {X 0,Y 419.945,Z 681.049,A -85,B 0,C 180,E1 20581.77,E2 20581.77} C_VEL
LIN {X 0,Y 421.614,Z 682.919,A -85,B 0,C 180,E1 20581.27,E2 20581.27} C_VEL
LIN {X 0,Y 422.302,Z 685.741,A -85,B 0,C 180,E1 20580.798,E2 20580.798} C_VEL
LIN {X 0,Y 421.759,Z 692.911,A -85,B 0,C 180,E1 20579.965,E2 20579.965} C_VEL
LIN {X 0,Y 420.132,Z 701.31,A -85,B 0,C 180,E1 20579.038,E2 20579.038} C_VEL
LIN {X 0,Y 420.573,Z 704.383,A -85,B 0,C 180,E1 20578.552,E2 20578.552} C_VEL
LIN {X 0,Y 428.054,Z 722.756,A -85,B 0,C 180,E1 20575.256,E2 20575.256} C_VEL
LIN {X 0,Y 434.886,Z 740.858,A -85,B 0,C 180,E1 20572.273,E2 20572.273} C_VEL
LIN {X 0,Y 441.705,Z 760.981,A -85,B 0,C 180,E1 20569.229,E2 20569.229} C_VEL
LIN {X 0,Y 444.296,Z 769.631,A -85,B 0,C 180,E1 20568.008,E2 20568.008} C_VEL
LIN {X 0,Y 438.26,Z 812.112,A -85,B 0,C 180,E1 20563.914,E2 20563.914} C_VEL
LIN {X 0,Y 432.523,Z 856.736,A -85,B 0,C 180,E1 20559.647,E2 20559.647} C_VEL
LIN {X 0,Y 427.332,Z 902.497,A -85,B 0,C 180,E1 20555.306,E2 20555.306} C_VEL
LIN {X 0,Y 426.007,Z 916.346,A -85,B 0,C 180,E1 20554.032,E2 20554.032} C_VEL
LIN {X 0,Y 426.686,Z 928.648,A -85,B 0,C 180,E1 20553.641,E2 20553.641} C_VEL
LIN {X 0,Y 421.271,Z 1023.322,A -85,B 0,C 180,E1 20551.047,E2 20551.047} C_VEL
LIN {X 0,Y 419.312,Z 1066.756,A -85,B 0,C 180,E1 20549.699,E2 20549.699} C_VEL
LIN {X 0,Y 418.394,Z 1084.764,A -85,B 0,C 180,E1 20548.865,E2 20548.865} C_VEL
LIN {X 0,Y 417.3,Z 1100.714,A -85,B 0,C 180,E1 20547.855,E2 20547.855} C_VEL
LIN {X 0,Y 416.032,Z 1116.031,A -85,B 0,C 180,E1 20546.618,E2 20546.618} C_VEL
LIN {X 0,Y 414.634,Z 1131.349,A -85,B 0,C 180,E1 20545.038,E2 20545.038} C_VEL
LIN {X 0,Y 413.352,Z 1144.321,A -85,B 0,C 180,E1 20543.373,E2 20543.373} C_VEL
LIN {X 0,Y 412.159,Z 1156.238,A -85,B 0,C 180,E1 20541.489,E2 20541.489} C_VEL
LIN {X 0,Y 411.169,Z 1166.486,A -85,B 0,C 180,E1 20539.461,E2 20539.461} C_VEL
LIN {X 0,Y 410.444,Z 1175.211,A -85,B 0,C 180,E1 20537.29,E2 20537.29} C_VEL
LIN {X 0,Y 409.977,Z 1182.247,A -85,B 0,C 180,E1 20534.983,E2 20534.983} C_VEL
LIN {X 0,Y 409.808,Z 1187.306,A -85,B 0,C 180,E1 20532.685,E2 20532.685} C_VEL
LIN {X 0,Y 409.899,Z 1190.713,A -85,B 0,C 180,E1 20530.258,E2 20530.258} C_VEL
LIN {X 0,Y 410.238,Z 1192.176,A -85,B 0,C 180,E1 20527.986,E2 20527.986} C_VEL
LIN {X 0,Y 410.971,Z 1191.898,A -85,B 0,C 180,E1 20525.445,E2 20525.445} C_VEL
LIN {X 0,Y 412.043,Z 1189.723,A -85,B 0,C 180,E1 20523.06,E2 20523.06} C_VEL
LIN {X 0,Y 413.577,Z 1185.766,A -85,B 0,C 180,E1 20520.693,E2 20520.693} C_VEL
LIN {X 0,Y 415.752,Z 1179.439,A -85,B 0,C 180,E1 20518.208,E2 20518.208} C_VEL
LIN {X 0,Y 418.182,Z 1171.722,A -85,B 0,C 180,E1 20516.024,E2 20516.024} C_VEL
LIN {X 0,Y 420.907,Z 1162.552,A -85,B 0,C 180,E1 20514,E2 20514} C_VEL
LIN {X 0,Y 424.063,Z 1151.07,A -85,B 0,C 180,E1 20512.003,E2 20512.003} C_VEL
LIN {X 0,Y 427.366,Z 1137.606,A -85,B 0,C 180,E1 20510.166,E2 20510.166} C_VEL
LIN {X 0,Y 430.389,Z 1123.995,A -85,B 0,C 180,E1 20508.679,E2 20508.679} C_VEL
LIN {X 0,Y 433.099,Z 1110.211,A -85,B 0,C 180,E1 20507.466,E2 20507.466} C_VEL
LIN {X 0,Y 435.95,Z 1092.886,A -85,B 0,C 180,E1 20506.268,E2 20506.268} C_VEL
LIN {X 0,Y 438.724,Z 1072.678,A -85,B 0,C 180,E1 20505.211,E2 20505.211} C_VEL
LIN {X 0,Y 444.901,Z 1035.682,A -85,B 0,C 180,E1 20503.583,E2 20503.583} C_VEL
LIN {X 0,Y 453.203,Z 986.896,A -85,B 0,C 180,E1 20501.751,E2 20501.751} C_VEL
LIN {X 0,Y 459,Z 947.582,A -85,B 0,C 180,E1 20500.465,E2 20500.465} C_VEL
LIN {X 0,Y 458.917,Z 943.016,A -85,B 0,C 180,E1 20500.129,E2 20500.129} C_VEL
LIN {X 0,Y 469.863,Z 910.483,A -85,B 0,C 180,E1 20496.417,E2 20496.417} C_VEL
LIN {X 0,Y 483.166,Z 878.574,A -85,B 0,C 180,E1 20492.65,E2 20492.65} C_VEL
LIN {X 0,Y 496.933,Z 851.959,A -85,B 0,C 180,E1 20489.398,E2 20489.398} C_VEL
LIN {X 0,Y 503.709,Z 840.749,A -85,B 0,C 180,E1 20487.994,E2 20487.994} C_VEL
LIN {X 0,Y 504.662,Z 838.96,A -85,B 0,C 180,E1 20486.521,E2 20486.521} C_VEL
LIN {X 0,Y 504.886,Z 838.761,A -85,B 0,C 180,E1 20486.186,E2 20486.186} C_VEL
LIN {X 0,Y 491.383,Z 861.366,A -85,B 0,C 180,E1 20483.782,E2 20483.782} C_VEL
LIN {X 0,Y 482.254,Z 880.728,A -85,B 0,C 180,E1 20481.537,E2 20481.537} C_VEL
LIN {X 0,Y 476.094,Z 898.698,A -85,B 0,C 180,E1 20479.299,E2 20479.299} C_VEL
LIN {X 0,Y 472.463,Z 916.029,A -85,B 0,C 180,E1 20476.983,E2 20476.983} C_VEL
LIN {X 0,Y 471.492,Z 933.227,A -85,B 0,C 180,E1 20474.58,E2 20474.58} C_VEL
LIN {X 0,Y 473.143,Z 949.416,A -85,B 0,C 180,E1 20472.221,E2 20472.221} C_VEL
LIN {X 0,Y 474.091,Z 954.74,A -85,B 0,C 180,E1 20471.468,E2 20471.468} C_VEL
LIN {X 0,Y 462.884,Z 977.464,A -85,B 0,C 180,E1 20470.472,E2 20470.472} C_VEL
LIN {X 0,Y 457.904,Z 989.394,A -85,B 0,C 180,E1 20469.891,E2 20469.891} C_VEL
LIN {X 0,Y 452.44,Z 1026.837,A -85,B 0,C 180,E1 20469.281,E2 20469.281} C_VEL
LIN {X 0,Y 449.076,Z 1051.68,A -85,B 0,C 180,E1 20468.554,E2 20468.554} C_VEL
LIN {X 0,Y 445.255,Z 1075.224,A -85,B 0,C 180,E1 20467.646,E2 20467.646} C_VEL
LIN {X 0,Y 440.799,Z 1099.233,A -85,B 0,C 180,E1 20466.461,E2 20466.461} C_VEL
LIN {X 0,Y 436.423,Z 1121.287,A -85,B 0,C 180,E1 20465.101,E2 20465.101} C_VEL
LIN {X 0,Y 431.478,Z 1144.959,A -85,B 0,C 180,E1 20463.31,E2 20463.31} C_VEL
LIN {X 0,Y 427.151,Z 1165.149,A -85,B 0,C 180,E1 20461.464,E2 20461.464} C_VEL
LIN {X 0,Y 422.995,Z 1184.425,A -85,B 0,C 180,E1 20459.37,E2 20459.37} C_VEL
LIN {X 0,Y 419.261,Z 1202.084,A -85,B 0,C 180,E1 20457.095,E2 20457.095} C_VEL
LIN {X 0,Y 414.647,Z 1228.18,A -85,B 0,C 180,E1 20453.293,E2 20453.293} C_VEL
LIN {X 0,Y 412.393,Z 1243.007,A -85,B 0,C 180,E1 20450.729,E2 20450.729} C_VEL
LIN {X 0,Y 410.797,Z 1254.919,A -85,B 0,C 180,E1 20448.297,E2 20448.297} C_VEL
LIN {X 0,Y 409.513,Z 1266.019,A -85,B 0,C 180,E1 20445.578,E2 20445.578} C_VEL
LIN {X 0,Y 408.735,Z 1275.088,A -85,B 0,C 180,E1 20442.86,E2 20442.86} C_VEL
LIN {X 0,Y 408.325,Z 1282.716,A -85,B 0,C 180,E1 20440.01,E2 20440.01} C_VEL
LIN {X 0,Y 408.223,Z 1288.378,A -85,B 0,C 180,E1 20437.252,E2 20437.252} C_VEL
LIN {X 0,Y 408.247,Z 1292.275,A -85,B 0,C 180,E1 20434.493,E2 20434.493} C_VEL
LIN {X 0,Y 408.305,Z 1294.671,A -85,B 0,C 180,E1 20431.682,E2 20431.682} C_VEL
LIN {X 0,Y 408.296,Z 1295.362,A -85,B 0,C 180,E1 20429.156,E2 20429.156} C_VEL
LIN {X 0,Y 408.201,Z 1294.602,A -85,B 0,C 180,E1 20426.347,E2 20426.347} C_VEL
LIN {X 0,Y 408.134,Z 1292.383,A -85,B 0,C 180,E1 20423.669,E2 20423.669} C_VEL
LIN {X 0,Y 408.213,Z 1288.375,A -85,B 0,C 180,E1 20420.796,E2 20420.796} C_VEL
LIN {X 0,Y 408.605,Z 1282.947,A -85,B 0,C 180,E1 20417.993,E2 20417.993} C_VEL
LIN {X 0,Y 409.462,Z 1275.626,A -85,B 0,C 180,E1 20415.141,E2 20415.141} C_VEL
LIN {X 0,Y 411.011,Z 1266.044,A -85,B 0,C 180,E1 20412.148,E2 20412.148} C_VEL
LIN {X 0,Y 413.197,Z 1254.959,A -85,B 0,C 180,E1 20409.309,E2 20409.309} C_VEL
LIN {X 0,Y 416,Z 1242.456,A -85,B 0,C 180,E1 20406.633,E2 20406.633} C_VEL
LIN {X 0,Y 419.577,Z 1227.736,A -85,B 0,C 180,E1 20403.991,E2 20403.991} C_VEL
LIN {X 0,Y 423.735,Z 1211.577,A -85,B 0,C 180,E1 20401.531,E2 20401.531} C_VEL
LIN {X 0,Y 428.731,Z 1192.848,A -85,B 0,C 180,E1 20399.122,E2 20399.122} C_VEL
LIN {X 0,Y 434.028,Z 1173.226,A -85,B 0,C 180,E1 20396.989,E2 20396.989} C_VEL
LIN {X 0,Y 439.814,Z 1151.961,A -85,B 0,C 180,E1 20395.045,E2 20395.045} C_VEL
LIN {X 0,Y 445.747,Z 1130.001,A -85,B 0,C 180,E1 20393.366,E2 20393.366} C_VEL
LIN {X 0,Y 451.946,Z 1106.514,A -85,B 0,C 180,E1 20391.882,E2 20391.882} C_VEL
LIN {X 0,Y 458.134,Z 1082.225,A -85,B 0,C 180,E1 20390.651,E2 20390.651} C_VEL
LIN {X 0,Y 464.431,Z 1055.563,A -85,B 0,C 180,E1 20389.595,E2 20389.595} C_VEL
LIN {X 0,Y 469.739,Z 1030.129,A -85,B 0,C 180,E1 20388.815,E2 20388.815} C_VEL
LIN {X 0,Y 476.523,Z 998.641,A -85,B 0,C 180,E1 20388.198,E2 20388.198} C_VEL
LIN {X 0,Y 484.068,Z 966.772,A -85,B 0,C 180,E1 20387.77,E2 20387.77} C_VEL
LIN {X 0,Y 486.547,Z 956.556,A -85,B 0,C 180,E1 20387.657,E2 20387.657} C_VEL
LIN {X 0,Y 487.057,Z 944.704,A -85,B 0,C 180,E1 20385.917,E2 20385.917} C_VEL
LIN {X 0,Y 489.679,Z 932.684,A -85,B 0,C 180,E1 20384.34,E2 20384.34} C_VEL
LIN {X 0,Y 491.525,Z 927.139,A -85,B 0,C 180,E1 20383.527,E2 20383.527} C_VEL
LIN {X 0,Y 476.65,Z 993.1,A -85,B 0,C 180,E1 20381.641,E2 20381.641} C_VEL
LIN {X 0,Y 468.418,Z 1034.362,A -85,B 0,C 180,E1 20380.38,E2 20380.38} C_VEL
LIN {X 0,Y 463.12,Z 1058.372,A -85,B 0,C 180,E1 20379.381,E2 20379.381} C_VEL
LIN {X 0,Y 457.395,Z 1081.851,A -85,B 0,C 180,E1 20378.138,E2 20378.138} C_VEL
LIN {X 0,Y 451.658,Z 1103.833,A -85,B 0,C 180,E1 20376.708,E2 20376.708} C_VEL
LIN {X 0,Y 445.622,Z 1125.717,A -85,B 0,C 180,E1 20374.98,E2 20374.98} C_VEL
LIN {X 0,Y 439.844,Z 1145.901,A -85,B 0,C 180,E1 20373.065,E2 20373.065} C_VEL
LIN {X 0,Y 434.34,Z 1164.516,A -85,B 0,C 180,E1 20370.965,E2 20370.965} C_VEL
LIN {X 0,Y 429.196,Z 1181.521,A -85,B 0,C 180,E1 20368.68,E2 20368.68} C_VEL
LIN {X 0,Y 424.579,Z 1196.55,A -85,B 0,C 180,E1 20366.279,E2 20366.279} C_VEL
LIN {X 0,Y 420.448,Z 1210.145,A -85,B 0,C 180,E1 20363.698,E2 20363.698} C_VEL
LIN {X 0,Y 416.861,Z 1222.234,A -85,B 0,C 180,E1 20360.94,E2 20360.94} C_VEL
LIN {X 0,Y 414.024,Z 1232.323,A -85,B 0,C 180,E1 20358.152,E2 20358.152} C_VEL
LIN {X 0,Y 411.777,Z 1240.95,A -85,B 0,C 180,E1 20355.204,E2 20355.204} C_VEL
LIN {X 0,Y 410.182,Z 1247.607,A -85,B 0,C 180,E1 20352.244,E2 20352.244} C_VEL
LIN {X 0,Y 409.152,Z 1252.54,A -85,B 0,C 180,E1 20349.282,E2 20349.282} C_VEL
LIN {X 0,Y 408.573,Z 1255.844,A -85,B 0,C 180,E1 20346.323,E2 20346.323} C_VEL
LIN {X 0,Y 408.277,Z 1257.421,A -85,B 0,C 180,E1 20343.51,E2 20343.51} C_VEL
LIN {X 0,Y 408.161,Z 1257.47,A -85,B 0,C 180,E1 20340.561,E2 20340.561} C_VEL
LIN {X 0,Y 408.125,Z 1256.043,A -85,B 0,C 180,E1 20337.753,E2 20337.753} C_VEL
LIN {X 0,Y 408.186,Z 1253.003,A -85,B 0,C 180,E1 20334.941,E2 20334.941} C_VEL
LIN {X 0,Y 408.404,Z 1248.403,A -85,B 0,C 180,E1 20332.12,E2 20332.12} C_VEL
LIN {X 0,Y 408.859,Z 1242.181,A -85,B 0,C 180,E1 20329.288,E2 20329.288} C_VEL
LIN {X 0,Y 409.636,Z 1234.52,A -85,B 0,C 180,E1 20326.592,E2 20326.592} C_VEL
LIN {X 0,Y 410.806,Z 1225.099,A -85,B 0,C 180,E1 20323.89,E2 20323.89} C_VEL
LIN {X 0,Y 412.453,Z 1213.744,A -85,B 0,C 180,E1 20321.19,E2 20321.19} C_VEL
LIN {X 0,Y 414.542,Z 1200.735,A -85,B 0,C 180,E1 20318.601,E2 20318.601} C_VEL
LIN {X 0,Y 416.917,Z 1186.58,A -85,B 0,C 180,E1 20316.239,E2 20316.239} C_VEL
LIN {X 0,Y 419.628,Z 1170.803,A -85,B 0,C 180,E1 20313.996,E2 20313.996} C_VEL
LIN {X 0,Y 422.696,Z 1152.939,A -85,B 0,C 180,E1 20311.841,E2 20311.841} C_VEL
LIN {X 0,Y 425.709,Z 1134.75,A -85,B 0,C 180,E1 20309.981,E2 20309.981} C_VEL
LIN {X 0,Y 428.815,Z 1114.992,A -85,B 0,C 180,E1 20308.277,E2 20308.277} C_VEL
LIN {X 0,Y 431.771,Z 1094.327,A -85,B 0,C 180,E1 20306.799,E2 20306.799} C_VEL
LIN {X 0,Y 434.387,Z 1073.874,A -85,B 0,C 180,E1 20305.59,E2 20305.59} C_VEL
LIN {X 0,Y 436.936,Z 1051.027,A -85,B 0,C 180,E1 20304.501,E2 20304.501} C_VEL
LIN {X 0,Y 439.001,Z 1028.474,A -85,B 0,C 180,E1 20303.667,E2 20303.667} C_VEL
LIN {X 0,Y 440.68,Z 1004.657,A -85,B 0,C 180,E1 20303.029,E2 20303.029} C_VEL
LIN {X 0,Y 454.426,Z 771.407,A -85,B 0,C 180,E1 20298.181,E2 20298.181} C_VEL
LIN {X 0,Y 438.419,Z 740.02,A -85,B 0,C 180,E1 20295.878,E2 20295.878} C_VEL
LIN {X 0,Y 421.818,Z 709.647,A -85,B 0,C 180,E1 20293.304,E2 20293.304} C_VEL
LIN {X 0,Y 414.643,Z 691.694,A -85,B 0,C 180,E1 20290.357,E2 20290.357} C_VEL
LIN {X 0,Y 410.612,Z 681.599,A -85,B 0,C 180,E1 20288.646,E2 20288.646} C_VEL
LIN {X 0,Y 410.596,Z 681.516,A -85,B 0,C 180,E1 20284.741,E2 20284.741} C_VEL
LIN {X 0,Y 410.612,Z 681.508,A -85,B 0,C 180,E1 20280.92,E2 20280.92} C_VEL
LIN {X 0,Y 410.602,Z 681.523,A -85,B 0,C 180,E1 20276.934,E2 20276.934} C_VEL
LIN {X 0,Y 410.61,Z 681.522,A -85,B 0,C 180,E1 20273.003,E2 20273.003} C_VEL
LIN {X 0,Y 410.598,Z 681.518,A -85,B 0,C 180,E1 20269.047,E2 20269.047} C_VEL
LIN {X 0,Y 410.596,Z 681.524,A -85,B 0,C 180,E1 20265.105,E2 20265.105} C_VEL
LIN {X 0,Y 410.604,Z 681.52,A -85,B 0,C 180,E1 20261.236,E2 20261.236} C_VEL
LIN {X 0,Y 410.61,Z 681.513,A -85,B 0,C 180,E1 20257.277,E2 20257.277} C_VEL
LIN {X 0,Y 410.594,Z 681.512,A -85,B 0,C 180,E1 20253.352,E2 20253.352} C_VEL
LIN {X 0,Y 410.593,Z 681.51,A -85,B 0,C 180,E1 20249.444,E2 20249.444} C_VEL
LIN {X 0,Y 410.604,Z 681.509,A -85,B 0,C 180,E1 20245.533,E2 20245.533} C_VEL
LIN {X 0,Y 410.603,Z 681.513,A -85,B 0,C 180,E1 20241.6,E2 20241.6} C_VEL
LIN {X 0,Y 410.606,Z 681.521,A -85,B 0,C 180,E1 20237.628,E2 20237.628} C_VEL
LIN {X 0,Y 410.595,Z 681.524,A -85,B 0,C 180,E1 20233.739,E2 20233.739} C_VEL
LIN {X 0,Y 410.596,Z 681.516,A -85,B 0,C 180,E1 20229.772,E2 20229.772} C_VEL
LIN {X 0,Y 410.605,Z 681.523,A -85,B 0,C 180,E1 20225.854,E2 20225.854} C_VEL
LIN {X 0,Y 410.64,Z 681.746,A -85,B 0,C 180,E1 20223.073,E2 20223.073} C_VEL
LIN {X 0,Y 411.991,Z 685.121,A -85,B 0,C 180,E1 20222.386,E2 20222.386} C_VEL
LIN {X 0,Y 417.987,Z 698.466,A -85,B 0,C 180,E1 20219.688,E2 20219.688} C_VEL
LIN {X 0,Y 420.573,Z 704.383,A -85,B 0,C 180,E1 20218.552,E2 20218.552} C_VEL
LIN {X 0,Y 421.735,Z 709.331,A -85,B 0,C 180,E1 20217.756,E2 20217.756} C_VEL
LIN {X 0,Y 421.639,Z 725.696,A -85,B 0,C 180,E1 20215.67,E2 20215.67} C_VEL
LIN {X 0,Y 422.484,Z 729.346,A -85,B 0,C 180,E1 20215.107,E2 20215.107} C_VEL
LIN {X 0,Y 429.283,Z 747.856,A -85,B 0,C 180,E1 20212.058,E2 20212.058} C_VEL
LIN {X 0,Y 436.005,Z 768.195,A -85,B 0,C 180,E1 20208.982,E2 20208.982} C_VEL
LIN {X 0,Y 437.258,Z 772.263,A -85,B 0,C 180,E1 20208.397,E2 20208.397} C_VEL
LIN {X 0,Y 431.075,Z 814.512,A -85,B 0,C 180,E1 20204.281,E2 20204.281} C_VEL
LIN {X 0,Y 425.233,Z 858.527,A -85,B 0,C 180,E1 20200.023,E2 20200.023} C_VEL
LIN {X 0,Y 419.845,Z 904.431,A -85,B 0,C 180,E1 20195.612,E2 20195.612} C_VEL
LIN {X 0,Y 418.598,Z 916.976,A -85,B 0,C 180,E1 20194.44,E2 20194.44} C_VEL
LIN {X 0,Y 419.236,Z 929.373,A -85,B 0,C 180,E1 20194.033,E2 20194.033} C_VEL
LIN {X 0,Y 413.91,Z 1019.305,A -85,B 0,C 180,E1 20191.512,E2 20191.512} C_VEL
LIN {X 0,Y 411.641,Z 1066.697,A -85,B 0,C 180,E1 20190.015,E2 20190.015} C_VEL
LIN {X 0,Y 410.702,Z 1084.516,A -85,B 0,C 180,E1 20189.178,E2 20189.178} C_VEL
LIN {X 0,Y 409.612,Z 1100.141,A -85,B 0,C 180,E1 20188.187,E2 20188.187} C_VEL
LIN {X 0,Y 408.306,Z 1115.503,A -85,B 0,C 180,E1 20186.939,E2 20186.939} C_VEL
LIN {X 0,Y 406.975,Z 1129.937,A -85,B 0,C 180,E1 20185.465,E2 20185.465} C_VEL
LIN {X 0,Y 405.627,Z 1143.43,A -85,B 0,C 180,E1 20183.762,E2 20183.762} C_VEL
LIN {X 0,Y 404.416,Z 1155.184,A -85,B 0,C 180,E1 20181.922,E2 20181.922} C_VEL
LIN {X 0,Y 403.355,Z 1165.901,A -85,B 0,C 180,E1 20179.853,E2 20179.853} C_VEL
LIN {X 0,Y 402.567,Z 1174.934,A -85,B 0,C 180,E1 20177.639,E2 20177.639} C_VEL
LIN {X 0,Y 402.079,Z 1181.933,A -85,B 0,C 180,E1 20175.432,E2 20175.432} C_VEL
LIN {X 0,Y 401.854,Z 1187.67,A -85,B 0,C 180,E1 20172.94,E2 20172.94} C_VEL
LIN {X 0,Y 401.911,Z 1191.192,A -85,B 0,C 180,E1 20170.609,E2 20170.609} C_VEL
LIN {X 0,Y 402.267,Z 1193.121,A -85,B 0,C 180,E1 20168.145,E2 20168.145} C_VEL
LIN {X 0,Y 402.947,Z 1193.165,A -85,B 0,C 180,E1 20165.696,E2 20165.696} C_VEL
LIN {X 0,Y 404.034,Z 1191.467,A -85,B 0,C 180,E1 20163.263,E2 20163.263} C_VEL
LIN {X 0,Y 405.567,Z 1187.896,A -85,B 0,C 180,E1 20160.848,E2 20160.848} C_VEL
LIN {X 0,Y 407.493,Z 1182.849,A -85,B 0,C 180,E1 20158.594,E2 20158.594} C_VEL
LIN {X 0,Y 410.25,Z 1174.942,A -85,B 0,C 180,E1 20156.087,E2 20156.087} C_VEL
LIN {X 0,Y 413.224,Z 1165.676,A -85,B 0,C 180,E1 20153.888,E2 20153.888} C_VEL
LIN {X 0,Y 416.233,Z 1155.511,A -85,B 0,C 180,E1 20151.991,E2 20151.991} C_VEL
LIN {X 0,Y 419.653,Z 1143.069,A -85,B 0,C 180,E1 20150.122,E2 20150.122} C_VEL
LIN {X 0,Y 423.013,Z 1129.293,A -85,B 0,C 180,E1 20148.478,E2 20148.478} C_VEL
LIN {X 0,Y 426.421,Z 1113.508,A -85,B 0,C 180,E1 20146.991,E2 20146.991} C_VEL
LIN {X 0,Y 429.257,Z 1098.027,A -85,B 0,C 180,E1 20145.843,E2 20145.843} C_VEL
LIN {X 0,Y 431.808,Z 1081.125,A -85,B 0,C 180,E1 20144.871,E2 20144.871} C_VEL
LIN {X 0,Y 437.298,Z 1048.838,A -85,B 0,C 180,E1 20143.336,E2 20143.336} C_VEL
LIN {X 0,Y 445.929,Z 1002.046,A -85,B 0,C 180,E1 20141.459,E2 20141.459} C_VEL
LIN {X 0,Y 452.776,Z 960.055,A -85,B 0,C 180,E1 20140.034,E2 20140.034} C_VEL
LIN {X 0,Y 454.259,Z 949.645,A -85,B 0,C 180,E1 20139.678,E2 20139.678} C_VEL
LIN {X 0,Y 454.149,Z 944.596,A -85,B 0,C 180,E1 20139.306,E2 20139.306} C_VEL
LIN {X 0,Y 466.272,Z 911.114,A -85,B 0,C 180,E1 20135.416,E2 20135.416} C_VEL
LIN {X 0,Y 479.867,Z 880.75,A -85,B 0,C 180,E1 20131.771,E2 20131.771} C_VEL
LIN {X 0,Y 494.297,Z 854.69,A -85,B 0,C 180,E1 20128.54,E2 20128.54} C_VEL
LIN {X 0,Y 499.434,Z 846.602,A -85,B 0,C 180,E1 20127.483,E2 20127.483} C_VEL
LIN {X 0,Y 500.053,Z 845.624,A -85,B 0,C 180,E1 20126.603,E2 20126.603} C_VEL
LIN {X 0,Y 487.135,Z 866.555,A -85,B 0,C 180,E1 20124.342,E2 20124.342} C_VEL
LIN {X 0,Y 477.727,Z 885.566,A -85,B 0,C 180,E1 20122.094,E2 20122.094} C_VEL
LIN {X 0,Y 470.98,Z 903.955,A -85,B 0,C 180,E1 20119.745,E2 20119.745} C_VEL
LIN {X 0,Y 467.211,Z 920.785,A -85,B 0,C 180,E1 20117.446,E2 20117.446} C_VEL
LIN {X 0,Y 465.896,Z 938.387,A -85,B 0,C 180,E1 20114.914,E2 20114.914} C_VEL
LIN {X 0,Y 467.281,Z 953.887,A -85,B 0,C 180,E1 20112.6,E2 20112.6} C_VEL
LIN {X 0,Y 467.693,Z 957.172,A -85,B 0,C 180,E1 20112.124,E2 20112.124} C_VEL
LIN {X 0,Y 456.763,Z 979.413,A -85,B 0,C 180,E1 20111.131,E2 20111.131} C_VEL
LIN {X 0,Y 453.106,Z 988.017,A -85,B 0,C 180,E1 20110.707,E2 20110.707} C_VEL
LIN {X 0,Y 447.329,Z 1026.46,A -85,B 0,C 180,E1 20110.069,E2 20110.069} C_VEL
LIN {X 0,Y 443.945,Z 1050.063,A -85,B 0,C 180,E1 20109.375,E2 20109.375} C_VEL
LIN {X 0,Y 439.817,Z 1073.945,A -85,B 0,C 180,E1 20108.443,E2 20108.443} C_VEL
LIN {X 0,Y 435.18,Z 1097.834,A -85,B 0,C 180,E1 20107.257,E2 20107.257} C_VEL
LIN {X 0,Y 430.56,Z 1119.669,A -85,B 0,C 180,E1 20105.898,E2 20105.898} C_VEL
LIN {X 0,Y 425.509,Z 1142.524,A -85,B 0,C 180,E1 20104.165,E2 20104.165} C_VEL
LIN {X 0,Y 420.906,Z 1162.795,A -85,B 0,C 180,E1 20102.307,E2 20102.307} C_VEL
LIN {X 0,Y 416.609,Z 1181.606,A -85,B 0,C 180,E1 20100.263,E2 20100.263} C_VEL
LIN {X 0,Y 412.43,Z 1199.958,A -85,B 0,C 180,E1 20097.896,E2 20097.896} C_VEL
LIN {X 0,Y 408.822,Z 1216.616,A -85,B 0,C 180,E1 20095.339,E2 20095.339} C_VEL
LIN {X 0,Y 405.527,Z 1235.991,A -85,B 0,C 180,E1 20092.161,E2 20092.161} C_VEL
LIN {X 0,Y 403.516,Z 1249.553,A -85,B 0,C 180,E1 20089.541,E2 20089.541} C_VEL
LIN {X 0,Y 402.067,Z 1261.008,A -85,B 0,C 180,E1 20086.913,E2 20086.913} C_VEL
LIN {X 0,Y 401.041,Z 1270.97,A -85,B 0,C 180,E1 20084.14,E2 20084.14} C_VEL
LIN {X 0,Y 400.471,Z 1279.013,A -85,B 0,C 180,E1 20081.374,E2 20081.374} C_VEL
LIN {X 0,Y 400.251,Z 1285.376,A -85,B 0,C 180,E1 20078.618,E2 20078.618} C_VEL
LIN {X 0,Y 400.235,Z 1289.805,A -85,B 0,C 180,E1 20076.021,E2 20076.021} C_VEL
LIN {X 0,Y 400.296,Z 1293.122,A -85,B 0,C 180,E1 20073.148,E2 20073.148} C_VEL
LIN {X 0,Y 400.322,Z 1294.662,A -85,B 0,C 180,E1 20070.57,E2 20070.57} C_VEL
LIN {X 0,Y 400.259,Z 1294.782,A -85,B 0,C 180,E1 20067.707,E2 20067.707} C_VEL
LIN {X 0,Y 400.16,Z 1293.431,A -85,B 0,C 180,E1 20064.981,E2 20064.981} C_VEL
LIN {X 0,Y 400.15,Z 1290.359,A -85,B 0,C 180,E1 20062.099,E2 20062.099} C_VEL
LIN {X 0,Y 400.383,Z 1285.758,A -85,B 0,C 180,E1 20059.203,E2 20059.203} C_VEL
LIN {X 0,Y 401.063,Z 1279.427,A -85,B 0,C 180,E1 20056.298,E2 20056.298} C_VEL
LIN {X 0,Y 402.371,Z 1270.921,A -85,B 0,C 180,E1 20053.244,E2 20053.244} C_VEL
LIN {X 0,Y 404.331,Z 1260.973,A -85,B 0,C 180,E1 20050.345,E2 20050.345} C_VEL
LIN {X 0,Y 407.11,Z 1248.938,A -85,B 0,C 180,E1 20047.441,E2 20047.441} C_VEL
LIN {X 0,Y 410.676,Z 1234.858,A -85,B 0,C 180,E1 20044.625,E2 20044.625} C_VEL
LIN {X 0,Y 414.713,Z 1219.989,A -85,B 0,C 180,E1 20042.111,E2 20042.111} C_VEL
LIN {X 0,Y 419.701,Z 1202.442,A -85,B 0,C 180,E1 20039.59,E2 20039.59} C_VEL
LIN {X 0,Y 425.3,Z 1183.232,A -85,B 0,C 180,E1 20037.265,E2 20037.265} C_VEL
LIN {X 0,Y 431.206,Z 1163.214,A -85,B 0,C 180,E1 20035.218,E2 20035.218} C_VEL
LIN {X 0,Y 437.756,Z 1140.985,A -85,B 0,C 180,E1 20033.314,E2 20033.314} C_VEL
LIN {X 0,Y 444.433,Z 1118.141,A -85,B 0,C 180,E1 20031.695,E2 20031.695} C_VEL
LIN {X 0,Y 451.407,Z 1093.559,A -85,B 0,C 180,E1 20030.278,E2 20030.278} C_VEL
LIN {X 0,Y 458.356,Z 1067.859,A -85,B 0,C 180,E1 20029.121,E2 20029.121} C_VEL
LIN {X 0,Y 465.056,Z 1040.092,A -85,B 0,C 180,E1 20028.149,E2 20028.149} C_VEL
LIN {X 0,Y 470.062,Z 1017.71,A -85,B 0,C 180,E1 20027.609,E2 20027.609} C_VEL
LIN {X 0,Y 478.214,Z 983.296,A -85,B 0,C 180,E1 20027.033,E2 20027.033} C_VEL
LIN {X 0,Y 483.945,Z 960.24,A -85,B 0,C 180,E1 20026.769,E2 20026.769} C_VEL
LIN {X 0,Y 485.388,Z 949.078,A -85,B 0,C 180,E1 20025.109,E2 20025.109} C_VEL
LIN {X 0,Y 487.369,Z 941.607,A -85,B 0,C 180,E1 20024.077,E2 20024.077} C_VEL
LIN {X 0,Y 471.447,Z 1009.032,A -85,B 0,C 180,E1 20022.134,E2 20022.134} C_VEL
LIN {X 0,Y 465.176,Z 1037.71,A -85,B 0,C 180,E1 20021.21,E2 20021.21} C_VEL
LIN {X 0,Y 459.372,Z 1061.272,A -85,B 0,C 180,E1 20020.194,E2 20020.194} C_VEL
LIN {X 0,Y 453.248,Z 1083.989,A -85,B 0,C 180,E1 20018.956,E2 20018.956} C_VEL
LIN {X 0,Y 446.931,Z 1105.993,A -85,B 0,C 180,E1 20017.483,E2 20017.483} C_VEL
LIN {X 0,Y 440.54,Z 1127.224,A -85,B 0,C 180,E1 20015.764,E2 20015.764} C_VEL
LIN {X 0,Y 434.41,Z 1146.946,A -85,B 0,C 180,E1 20013.85,E2 20013.85} C_VEL
LIN {X 0,Y 428.383,Z 1165.746,A -85,B 0,C 180,E1 20011.68,E2 20011.68} C_VEL
LIN {X 0,Y 422.78,Z 1182.943,A -85,B 0,C 180,E1 20009.312,E2 20009.312} C_VEL
LIN {X 0,Y 417.604,Z 1198.604,A -85,B 0,C 180,E1 20006.733,E2 20006.733} C_VEL
LIN {X 0,Y 413.272,Z 1211.784,A -85,B 0,C 180,E1 20004.135,E2 20004.135} C_VEL
LIN {X 0,Y 409.646,Z 1223.063,A -85,B 0,C 180,E1 20001.477,E2 20001.477} C_VEL
LIN {X 0,Y 406.591,Z 1233.046,A -85,B 0,C 180,E1 19998.645,E2 19998.645} C_VEL
LIN {X 0,Y 404.161,Z 1241.597,A -85,B 0,C 180,E1 19995.644,E2 19995.644} C_VEL
LIN {X 0,Y 402.425,Z 1248.196,A -85,B 0,C 180,E1 19992.63,E2 19992.63} C_VEL
LIN {X 0,Y 401.284,Z 1253.076,A -85,B 0,C 180,E1 19989.61,E2 19989.61} C_VEL
LIN {X 0,Y 400.641,Z 1256.336,A -85,B 0,C 180,E1 19986.592,E2 19986.592} C_VEL
LIN {X 0,Y 400.31,Z 1257.883,A -85,B 0,C 180,E1 19983.724,E2 19983.724} C_VEL
LIN {X 0,Y 400.177,Z 1257.932,A -85,B 0,C 180,E1 19980.859,E2 19980.859} C_VEL
LIN {X 0,Y 400.133,Z 1256.559,A -85,B 0,C 180,E1 19977.995,E2 19977.995} C_VEL
LIN {X 0,Y 400.182,Z 1253.54,A -85,B 0,C 180,E1 19975.127,E2 19975.127} C_VEL
LIN {X 0,Y 400.409,Z 1248.713,A -85,B 0,C 180,E1 19972.106,E2 19972.106} C_VEL
LIN {X 0,Y 400.877,Z 1242.441,A -85,B 0,C 180,E1 19969.218,E2 19969.218} C_VEL
LIN {X 0,Y 401.679,Z 1234.734,A -85,B 0,C 180,E1 19966.468,E2 19966.468} C_VEL
LIN {X 0,Y 402.889,Z 1225.243,A -85,B 0,C 180,E1 19963.713,E2 19963.713} C_VEL
LIN {X 0,Y 404.593,Z 1213.807,A -85,B 0,C 180,E1 19960.96,E2 19960.96} C_VEL
LIN {X 0,Y 406.718,Z 1200.921,A -85,B 0,C 180,E1 19958.36,E2 19958.36} C_VEL
LIN {X 0,Y 409.378,Z 1185.583,A -85,B 0,C 180,E1 19955.774,E2 19955.774} C_VEL
LIN {X 0,Y 412.2,Z 1169.524,A -85,B 0,C 180,E1 19953.491,E2 19953.491} C_VEL
LIN {X 0,Y 415.284,Z 1151.963,A -85,B 0,C 180,E1 19951.371,E2 19951.371} C_VEL
LIN {X 0,Y 418.528,Z 1132.753,A -85,B 0,C 180,E1 19949.411,E2 19949.411} C_VEL
LIN {X 0,Y 421.613,Z 1113.448,A -85,B 0,C 180,E1 19947.75,E2 19947.75} C_VEL
LIN {X 0,Y 424.694,Z 1092.467,A -85,B 0,C 180,E1 19946.245,E2 19946.245} C_VEL
LIN {X 0,Y 427.56,Z 1070.282,A -85,B 0,C 180,E1 19944.953,E2 19944.953} C_VEL
LIN {X 0,Y 430.009,Z 1048.116,A -85,B 0,C 180,E1 19943.922,E2 19943.922} C_VEL
LIN {X 0,Y 432.13,Z 1024.461,A -85,B 0,C 180,E1 19943.077,E2 19943.077} C_VEL
LIN {X 0,Y 433.909,Z 998.156,A -85,B 0,C 180,E1 19942.414,E2 19942.414} C_VEL
LIN {X 0,Y 447.734,Z 774.144,A -85,B 0,C 180,E1 19937.665,E2 19937.665} C_VEL
LIN {X 0,Y 431.436,Z 742.217,A -85,B 0,C 180,E1 19935.264,E2 19935.264} C_VEL
LIN {X 0,Y 415.427,Z 713.112,A -85,B 0,C 180,E1 19932.747,E2 19932.747} C_VEL
LIN {X 0,Y 413.652,Z 709.733,A -85,B 0,C 180,E1 19932.41,E2 19932.41} C_VEL
LIN {X 0,Y 405.656,Z 689.904,A -85,B 0,C 180,E1 19929.064,E2 19929.064} C_VEL
LIN {X 0,Y 402.687,Z 682.647,A -85,B 0,C 180,E1 19927.792,E2 19927.792} C_VEL
LIN {X 0,Y 402.656,Z 682.502,A -85,B 0,C 180,E1 19923.798,E2 19923.798} C_VEL
LIN {X 0,Y 402.657,Z 682.506,A -85,B 0,C 180,E1 19919.78,E2 19919.78} C_VEL
LIN {X 0,Y 402.663,Z 682.509,A -85,B 0,C 180,E1 19915.917,E2 19915.917} C_VEL
LIN {X 0,Y 402.664,Z 682.51,A -85,B 0,C 180,E1 19912.024,E2 19912.024} C_VEL
LIN {X 0,Y 402.667,Z 682.512,A -85,B 0,C 180,E1 19908.085,E2 19908.085} C_VEL
LIN {X 0,Y 402.656,Z 682.503,A -85,B 0,C 180,E1 19904.087,E2 19904.087} C_VEL
LIN {X 0,Y 402.658,Z 682.51,A -85,B 0,C 180,E1 19900.157,E2 19900.157} C_VEL
LIN {X 0,Y 402.669,Z 682.51,A -85,B 0,C 180,E1 19896.274,E2 19896.274} C_VEL
LIN {X 0,Y 402.66,Z 682.511,A -85,B 0,C 180,E1 19892.279,E2 19892.279} C_VEL
LIN {X 0,Y 402.669,Z 682.508,A -85,B 0,C 180,E1 19888.437,E2 19888.437} C_VEL
LIN {X 0,Y 402.656,Z 682.512,A -85,B 0,C 180,E1 19884.444,E2 19884.444} C_VEL
LIN {X 0,Y 402.66,Z 682.511,A -85,B 0,C 180,E1 19880.569,E2 19880.569} C_VEL
LIN {X 0,Y 402.666,Z 682.507,A -85,B 0,C 180,E1 19876.504,E2 19876.504} C_VEL
LIN {X 0,Y 402.668,Z 682.504,A -85,B 0,C 180,E1 19872.466,E2 19872.466} C_VEL
LIN {X 0,Y 402.662,Z 682.514,A -85,B 0,C 180,E1 19868.44,E2 19868.44} C_VEL
LIN {X 0,Y 402.658,Z 682.507,A -85,B 0,C 180,E1 19864.403,E2 19864.403} C_VEL
LIN {X 0,Y 402.688,Z 682.703,A -85,B 0,C 180,E1 19864.189,E2 19864.189} C_VEL
LIN {X 0,Y 403.88,Z 685.854,A -85,B 0,C 180,E1 19863.539,E2 19863.539} C_VEL
LIN {X 0,Y 408.355,Z 695.464,A -85,B 0,C 180,E1 19861.482,E2 19861.482} C_VEL
LIN {X 0,Y 415.876,Z 712.834,A -85,B 0,C 180,E1 19858.069,E2 19858.069} C_VEL
LIN {X 0,Y 422.484,Z 729.346,A -85,B 0,C 180,E1 19855.107,E2 19855.107} C_VEL
LIN {X 0,Y 423.454,Z 734.579,A -85,B 0,C 180,E1 19854.342,E2 19854.342} C_VEL
LIN {X 0,Y 423.01,Z 751.408,A -85,B 0,C 180,E1 19852.337,E2 19852.337} C_VEL
LIN {X 0,Y 423.783,Z 755.196,A -85,B 0,C 180,E1 19851.793,E2 19851.793} C_VEL
LIN {X 0,Y 430.203,Z 775.228,A -85,B 0,C 180,E1 19848.764,E2 19848.764} C_VEL
LIN {X 0,Y 423.655,Z 818.442,A -85,B 0,C 180,E1 19844.505,E2 19844.505} C_VEL
LIN {X 0,Y 417.738,Z 861.777,A -85,B 0,C 180,E1 19840.261,E2 19840.261} C_VEL
LIN {X 0,Y 412.34,Z 906.415,A -85,B 0,C 180,E1 19835.916,E2 19835.916} C_VEL
LIN {X 0,Y 411.204,Z 917.755,A -85,B 0,C 180,E1 19834.853,E2 19834.853} C_VEL
LIN {X 0,Y 411.807,Z 930.098,A -85,B 0,C 180,E1 19834.438,E2 19834.438} C_VEL
LIN {X 0,Y 406.544,Z 1015.855,A -85,B 0,C 180,E1 19831.978,E2 19831.978} C_VEL
LIN {X 0,Y 403.957,Z 1066.282,A -85,B 0,C 180,E1 19830.338,E2 19830.338} C_VEL
LIN {X 0,Y 403.057,Z 1083.391,A -85,B 0,C 180,E1 19829.542,E2 19829.542} C_VEL
LIN {X 0,Y 401.876,Z 1100.218,A -85,B 0,C 180,E1 19828.478,E2 19828.478} C_VEL
LIN {X 0,Y 400.436,Z 1116.741,A -85,B 0,C 180,E1 19827.11,E2 19827.11} C_VEL
LIN {X 0,Y 399.14,Z 1130.45,A -85,B 0,C 180,E1 19825.683,E2 19825.683} C_VEL
LIN {X 0,Y 397.702,Z 1144.493,A -85,B 0,C 180,E1 19823.878,E2 19823.878} C_VEL
LIN {X 0,Y 396.419,Z 1156.682,A -85,B 0,C 180,E1 19821.919,E2 19821.919} C_VEL
LIN {X 0,Y 395.42,Z 1166.608,A -85,B 0,C 180,E1 19819.961,E2 19819.961} C_VEL
LIN {X 0,Y 394.607,Z 1175.692,A -85,B 0,C 180,E1 19817.694,E2 19817.694} C_VEL
LIN {X 0,Y 394.105,Z 1182.833,A -85,B 0,C 180,E1 19815.409,E2 19815.409} C_VEL
LIN {X 0,Y 393.89,Z 1188.535,A -85,B 0,C 180,E1 19812.907,E2 19812.907} C_VEL
LIN {X 0,Y 393.964,Z 1192.143,A -85,B 0,C 180,E1 19810.529,E2 19810.529} C_VEL
LIN {X 0,Y 394.35,Z 1194.14,A -85,B 0,C 180,E1 19808.016,E2 19808.016} C_VEL
LIN {X 0,Y 395.032,Z 1194.337,A -85,B 0,C 180,E1 19805.665,E2 19805.665} C_VEL
LIN {X 0,Y 396.247,Z 1192.679,A -85,B 0,C 180,E1 19803.038,E2 19803.038} C_VEL
LIN {X 0,Y 397.878,Z 1189.216,A -85,B 0,C 180,E1 19800.576,E2 19800.576} C_VEL
LIN {X 0,Y 400.064,Z 1183.926,A -85,B 0,C 180,E1 19798.138,E2 19798.138} C_VEL
LIN {X 0,Y 402.83,Z 1176.563,A -85,B 0,C 180,E1 19795.73,E2 19795.73} C_VEL
LIN {X 0,Y 405.741,Z 1168.093,A -85,B 0,C 180,E1 19793.633,E2 19793.633} C_VEL
LIN {X 0,Y 409.133,Z 1157.603,A -85,B 0,C 180,E1 19791.568,E2 19791.568} C_VEL
LIN {X 0,Y 412.704,Z 1145.408,A -85,B 0,C 180,E1 19789.672,E2 19789.672} C_VEL
LIN {X 0,Y 416.527,Z 1130.859,A -85,B 0,C 180,E1 19787.875,E2 19787.875} C_VEL
LIN {X 0,Y 419.954,Z 1116.099,A -85,B 0,C 180,E1 19786.436,E2 19786.436} C_VEL
LIN {X 0,Y 423.102,Z 1100.232,A -85,B 0,C 180,E1 19785.213,E2 19785.213} C_VEL
LIN {X 0,Y 425.748,Z 1084.598,A -85,B 0,C 180,E1 19784.261,E2 19784.261} C_VEL
LIN {X 0,Y 431.764,Z 1051.353,A -85,B 0,C 180,E1 19782.618,E2 19782.618} C_VEL
LIN {X 0,Y 440.586,Z 1006.138,A -85,B 0,C 180,E1 19780.757,E2 19780.757} C_VEL
LIN {X 0,Y 447.426,Z 966.797,A -85,B 0,C 180,E1 19779.379,E2 19779.379} C_VEL
LIN {X 0,Y 449.691,Z 951.858,A -85,B 0,C 180,E1 19778.878,E2 19778.878} C_VEL
LIN {X 0,Y 449.777,Z 945.941,A -85,B 0,C 180,E1 19778.413,E2 19778.413} C_VEL
LIN {X 0,Y 461.292,Z 915.752,A -85,B 0,C 180,E1 19774.859,E2 19774.859} C_VEL
LIN {X 0,Y 475.398,Z 885.69,A -85,B 0,C 180,E1 19771.207,E2 19771.207} C_VEL
LIN {X 0,Y 489.816,Z 860.74,A -85,B 0,C 180,E1 19768.081,E2 19768.081} C_VEL
LIN {X 0,Y 495.176,Z 852.69,A -85,B 0,C 180,E1 19767.016,E2 19767.016} C_VEL
LIN {X 0,Y 481.997,Z 873.512,A -85,B 0,C 180,E1 19764.712,E2 19764.712} C_VEL
LIN {X 0,Y 472.211,Z 892.815,A -85,B 0,C 180,E1 19762.362,E2 19762.362} C_VEL
LIN {X 0,Y 465.618,Z 910.387,A -85,B 0,C 180,E1 19760.049,E2 19760.049} C_VEL
LIN {X 0,Y 461.655,Z 927.736,A -85,B 0,C 180,E1 19757.606,E2 19757.606} C_VEL
LIN {X 0,Y 460.346,Z 944.77,A -85,B 0,C 180,E1 19755.076,E2 19755.076} C_VEL
LIN {X 0,Y 461.585,Z 959.613,A -85,B 0,C 180,E1 19752.813,E2 19752.813} C_VEL
LIN {X 0,Y 450.336,Z 982.505,A -85,B 0,C 180,E1 19751.763,E2 19751.763} C_VEL
LIN {X 0,Y 448.646,Z 986.786,A -85,B 0,C 180,E1 19751.566,E2 19751.566} C_VEL
LIN {X 0,Y 442.256,Z 1027.496,A -85,B 0,C 180,E1 19750.859,E2 19750.859} C_VEL
LIN {X 0,Y 438.577,Z 1051.114,A -85,B 0,C 180,E1 19750.135,E2 19750.135} C_VEL
LIN {X 0,Y 433.529,Z 1078.28,A -85,B 0,C 180,E1 19749.021,E2 19749.021} C_VEL
LIN {X 0,Y 428.923,Z 1100.066,A -85,B 0,C 180,E1 19747.877,E2 19747.877} C_VEL
LIN {X 0,Y 423.39,Z 1124.681,A -85,B 0,C 180,E1 19746.267,E2 19746.267} C_VEL
LIN {X 0,Y 418.366,Z 1145.753,A -85,B 0,C 180,E1 19744.566,E2 19744.566} C_VEL
LIN {X 0,Y 413.352,Z 1166.614,A -85,B 0,C 180,E1 19742.56,E2 19742.56} C_VEL
LIN {X 0,Y 408.357,Z 1186.959,A -85,B 0,C 180,E1 19740.192,E2 19740.192} C_VEL
LIN {X 0,Y 404.327,Z 1203.769,A -85,B 0,C 180,E1 19737.862,E2 19737.862} C_VEL
LIN {X 0,Y 400.678,Z 1219.725,A -85,B 0,C 180,E1 19735.258,E2 19735.258} C_VEL
LIN {X 0,Y 397.6,Z 1236.008,A -85,B 0,C 180,E1 19732.315,E2 19732.315} C_VEL
LIN {X 0,Y 395.548,Z 1249.52,A -85,B 0,C 180,E1 19729.643,E2 19729.643} C_VEL
LIN {X 0,Y 394.065,Z 1261,A -85,B 0,C 180,E1 19726.943,E2 19726.943} C_VEL
LIN {X 0,Y 393.036,Z 1270.869,A -85,B 0,C 180,E1 19724.134,E2 19724.134} C_VEL
LIN {X 0,Y 392.468,Z 1278.852,A -85,B 0,C 180,E1 19721.311,E2 19721.311} C_VEL
LIN {X 0,Y 392.258,Z 1285.422,A -85,B 0,C 180,E1 19718.352,E2 19718.352} C_VEL
LIN {X 0,Y 392.255,Z 1289.765,A -85,B 0,C 180,E1 19715.703,E2 19715.703} C_VEL
LIN {X 0,Y 392.323,Z 1292.898,A -85,B 0,C 180,E1 19712.774,E2 19712.774} C_VEL
LIN {X 0,Y 392.34,Z 1294.392,A -85,B 0,C 180,E1 19709.998,E2 19709.998} C_VEL
LIN {X 0,Y 392.257,Z 1294.263,A -85,B 0,C 180,E1 19707.222,E2 19707.222} C_VEL
LIN {X 0,Y 392.145,Z 1292.65,A -85,B 0,C 180,E1 19704.291,E2 19704.291} C_VEL
LIN {X 0,Y 392.177,Z 1289.548,A -85,B 0,C 180,E1 19701.494,E2 19701.494} C_VEL
LIN {X 0,Y 392.553,Z 1284.186,A -85,B 0,C 180,E1 19698.241,E2 19698.241} C_VEL
LIN {X 0,Y 393.431,Z 1277.63,A -85,B 0,C 180,E1 19695.275,E2 19695.275} C_VEL
LIN {X 0,Y 394.943,Z 1269.218,A -85,B 0,C 180,E1 19692.312,E2 19692.312} C_VEL
LIN {X 0,Y 397.327,Z 1258.474,A -85,B 0,C 180,E1 19689.215,E2 19689.215} C_VEL
LIN {X 0,Y 400.466,Z 1246.218,A -85,B 0,C 180,E1 19686.296,E2 19686.296} C_VEL
LIN {X 0,Y 404.372,Z 1232.379,A -85,B 0,C 180,E1 19683.524,E2 19683.524} C_VEL
LIN {X 0,Y 409.308,Z 1215.813,A -85,B 0,C 180,E1 19680.751,E2 19680.751} C_VEL
LIN {X 0,Y 414.706,Z 1198.348,A -85,B 0,C 180,E1 19678.289,E2 19678.289} C_VEL
LIN {X 0,Y 420.926,Z 1178.682,A -85,B 0,C 180,E1 19675.945,E2 19675.945} C_VEL
LIN {X 0,Y 427.733,Z 1157.443,A -85,B 0,C 180,E1 19673.823,E2 19673.823} C_VEL
LIN {X 0,Y 434.91,Z 1135.086,A -85,B 0,C 180,E1 19671.963,E2 19671.963} C_VEL
LIN {X 0,Y 442.489,Z 1111.218,A -85,B 0,C 180,E1 19670.329,E2 19670.329} C_VEL
LIN {X 0,Y 449.841,Z 1087.437,A -85,B 0,C 180,E1 19669.025,E2 19669.025} C_VEL
LIN {X 0,Y 456.986,Z 1062.936,A -85,B 0,C 180,E1 19667.968,E2 19667.968} C_VEL
LIN {X 0,Y 463.968,Z 1036.117,A -85,B 0,C 180,E1 19667.066,E2 19667.066} C_VEL
LIN {X 0,Y 471.229,Z 1006.07,A -85,B 0,C 180,E1 19666.426,E2 19666.426} C_VEL
LIN {X 0,Y 480.599,Z 968.981,A -85,B 0,C 180,E1 19665.918,E2 19665.918} C_VEL
LIN {X 0,Y 481.855,Z 964.03,A -85,B 0,C 180,E1 19665.856,E2 19665.856} C_VEL
LIN {X 0,Y 483.44,Z 956.078,A -85,B 0,C 180,E1 19664.637,E2 19664.637} C_VEL
LIN {X 0,Y 466.905,Z 1022.728,A -85,B 0,C 180,E1 19662.703,E2 19662.703} C_VEL
LIN {X 0,Y 461.569,Z 1044.28,A -85,B 0,C 180,E1 19661.936,E2 19661.936} C_VEL
LIN {X 0,Y 455.215,Z 1067.168,A -85,B 0,C 180,E1 19660.887,E2 19660.887} C_VEL
LIN {X 0,Y 448.257,Z 1090.198,A -85,B 0,C 180,E1 19659.557,E2 19659.557} C_VEL
LIN {X 0,Y 441.182,Z 1112.336,A -85,B 0,C 180,E1 19657.976,E2 19657.976} C_VEL
LIN {X 0,Y 434.321,Z 1132.99,A -85,B 0,C 180,E1 19656.194,E2 19656.194} C_VEL
LIN {X 0,Y 427.547,Z 1152.818,A -85,B 0,C 180,E1 19654.145,E2 19654.145} C_VEL
LIN {X 0,Y 421.156,Z 1171.113,A -85,B 0,C 180,E1 19651.887,E2 19651.887} C_VEL
LIN {X 0,Y 415.214,Z 1187.862,A -85,B 0,C 180,E1 19649.424,E2 19649.424} C_VEL
LIN {X 0,Y 409.809,Z 1203.068,A -85,B 0,C 180,E1 19646.745,E2 19646.745} C_VEL
LIN {X 0,Y 405.268,Z 1215.969,A -85,B 0,C 180,E1 19644.023,E2 19644.023} C_VEL
LIN {X 0,Y 401.431,Z 1227.196,A -85,B 0,C 180,E1 19641.172,E2 19641.172} C_VEL
LIN {X 0,Y 398.244,Z 1236.874,A -85,B 0,C 180,E1 19638.14,E2 19638.14} C_VEL
LIN {X 0,Y 395.954,Z 1244.284,A -85,B 0,C 180,E1 19635.226,E2 19635.226} C_VEL
LIN {X 0,Y 394.209,Z 1250.601,A -85,B 0,C 180,E1 19632.005,E2 19632.005} C_VEL
LIN {X 0,Y 393.153,Z 1254.931,A -85,B 0,C 180,E1 19628.925,E2 19628.925} C_VEL
LIN {X 0,Y 392.552,Z 1257.531,A -85,B 0,C 180,E1 19625.848,E2 19625.848} C_VEL
LIN {X 0,Y 392.259,Z 1258.52,A -85,B 0,C 180,E1 19622.776,E2 19622.776} C_VEL
LIN {X 0,Y 392.173,Z 1258.001,A -85,B 0,C 180,E1 19619.854,E2 19619.854} C_VEL
LIN {X 0,Y 392.137,Z 1255.878,A -85,B 0,C 180,E1 19616.931,E2 19616.931} C_VEL
LIN {X 0,Y 392.253,Z 1252.011,A -85,B 0,C 180,E1 19613.854,E2 19613.854} C_VEL
LIN {X 0,Y 392.574,Z 1246.713,A -85,B 0,C 180,E1 19610.914,E2 19610.914} C_VEL
LIN {X 0,Y 393.195,Z 1239.612,A -85,B 0,C 180,E1 19607.964,E2 19607.964} C_VEL
LIN {X 0,Y 394.207,Z 1230.939,A -85,B 0,C 180,E1 19605.107,E2 19605.107} C_VEL
LIN {X 0,Y 395.739,Z 1220.15,A -85,B 0,C 180,E1 19602.198,E2 19602.198} C_VEL
LIN {X 0,Y 397.654,Z 1208.338,A -85,B 0,C 180,E1 19599.542,E2 19599.542} C_VEL
LIN {X 0,Y 400.108,Z 1194.169,A -85,B 0,C 180,E1 19596.878,E2 19596.878} C_VEL
LIN {X 0,Y 402.808,Z 1179.087,A -85,B 0,C 180,E1 19594.489,E2 19594.489} C_VEL
LIN {X 0,Y 405.823,Z 1162.451,A -85,B 0,C 180,E1 19592.246,E2 19592.246} C_VEL
LIN {X 0,Y 409.041,Z 1144.351,A -85,B 0,C 180,E1 19590.176,E2 19590.176} C_VEL
LIN {X 0,Y 412.294,Z 1125.239,A -85,B 0,C 180,E1 19588.328,E2 19588.328} C_VEL
LIN {X 0,Y 415.582,Z 1104.356,A -85,B 0,C 180,E1 19586.64,E2 19586.64} C_VEL
LIN {X 0,Y 418.695,Z 1082.553,A -85,B 0,C 180,E1 19585.197,E2 19585.197} C_VEL
LIN {X 0,Y 421.37,Z 1060.9,A -85,B 0,C 180,E1 19584.034,E2 19584.034} C_VEL
LIN {X 0,Y 423.808,Z 1037.562,A -85,B 0,C 180,E1 19583.045,E2 19583.045} C_VEL
LIN {X 0,Y 425.798,Z 1013.813,A -85,B 0,C 180,E1 19582.299,E2 19582.299} C_VEL
LIN {X 0,Y 440.848,Z 776.581,A -85,B 0,C 180,E1 19577.122,E2 19577.122} C_VEL
LIN {X 0,Y 424.912,Z 745.338,A -85,B 0,C 180,E1 19574.718,E2 19574.718} C_VEL
LIN {X 0,Y 409.482,Z 717.225,A -85,B 0,C 180,E1 19572.232,E2 19572.232} C_VEL
LIN {X 0,Y 405.602,Z 710.196,A -85,B 0,C 180,E1 19571.541,E2 19571.541} C_VEL
LIN {X 0,Y 397.739,Z 690.877,A -85,B 0,C 180,E1 19568.203,E2 19568.203} C_VEL
LIN {X 0,Y 394.822,Z 684.129,A -85,B 0,C 180,E1 19566.977,E2 19566.977} C_VEL
LIN {X 0,Y 394.718,Z 683.493,A -85,B 0,C 180,E1 19566.823,E2 19566.823} C_VEL
LIN {X 0,Y 394.732,Z 683.499,A -85,B 0,C 180,E1 19562.755,E2 19562.755} C_VEL
LIN {X 0,Y 394.725,Z 683.5,A -85,B 0,C 180,E1 19558.772,E2 19558.772} C_VEL
LIN {X 0,Y 394.722,Z 683.501,A -85,B 0,C 180,E1 19554.708,E2 19554.708} C_VEL
LIN {X 0,Y 394.73,Z 683.499,A -85,B 0,C 180,E1 19550.773,E2 19550.773} C_VEL
LIN {X 0,Y 394.722,Z 683.497,A -85,B 0,C 180,E1 19546.757,E2 19546.757} C_VEL
LIN {X 0,Y 394.727,Z 683.483,A -85,B 0,C 180,E1 19542.733,E2 19542.733} C_VEL
LIN {X 0,Y 394.714,Z 683.484,A -85,B 0,C 180,E1 19538.744,E2 19538.744} C_VEL
LIN {X 0,Y 394.716,Z 683.491,A -85,B 0,C 180,E1 19534.797,E2 19534.797} C_VEL
LIN {X 0,Y 394.723,Z 683.492,A -85,B 0,C 180,E1 19530.728,E2 19530.728} C_VEL
LIN {X 0,Y 394.718,Z 683.492,A -85,B 0,C 180,E1 19526.807,E2 19526.807} C_VEL
LIN {X 0,Y 394.726,Z 683.49,A -85,B 0,C 180,E1 19522.872,E2 19522.872} C_VEL
LIN {X 0,Y 394.716,Z 683.489,A -85,B 0,C 180,E1 19518.902,E2 19518.902} C_VEL
LIN {X 0,Y 394.72,Z 683.496,A -85,B 0,C 180,E1 19514.878,E2 19514.878} C_VEL
LIN {X 0,Y 394.73,Z 683.5,A -85,B 0,C 180,E1 19510.883,E2 19510.883} C_VEL
LIN {X 0,Y 394.724,Z 683.495,A -85,B 0,C 180,E1 19506.858,E2 19506.858} C_VEL
LIN {X 0,Y 394.756,Z 683.678,A -85,B 0,C 180,E1 19505.358,E2 19505.358} C_VEL
LIN {X 0,Y 396.163,Z 687.176,A -85,B 0,C 180,E1 19504.594,E2 19504.594} C_VEL
LIN {X 0,Y 400.814,Z 697.375,A -85,B 0,C 180,E1 19502.357,E2 19502.357} C_VEL
LIN {X 0,Y 406.815,Z 710.847,A -85,B 0,C 180,E1 19499.584,E2 19499.584} C_VEL
LIN {X 0,Y 414.37,Z 729.457,A -85,B 0,C 180,E1 19496.108,E2 19496.108} C_VEL
LIN {X 0,Y 421.311,Z 748.105,A -85,B 0,C 180,E1 19492.931,E2 19492.931} C_VEL
LIN {X 0,Y 423.783,Z 755.196,A -85,B 0,C 180,E1 19491.793,E2 19491.793} C_VEL
LIN {X 0,Y 424.874,Z 761.356,A -85,B 0,C 180,E1 19490.938,E2 19490.938} C_VEL
LIN {X 0,Y 424.45,Z 769.946,A -85,B 0,C 180,E1 19489.969,E2 19489.969} C_VEL
LIN {X 0,Y 422.399,Z 782.605,A -85,B 0,C 180,E1 19488.699,E2 19488.699} C_VEL
LIN {X 0,Y 415.996,Z 824.005,A -85,B 0,C 180,E1 19484.576,E2 19484.576} C_VEL
LIN {X 0,Y 410.147,Z 865.853,A -85,B 0,C 180,E1 19480.427,E2 19480.427} C_VEL
LIN {X 0,Y 404.703,Z 909.604,A -85,B 0,C 180,E1 19476.112,E2 19476.112} C_VEL
LIN {X 0,Y 403.808,Z 918.467,A -85,B 0,C 180,E1 19475.276,E2 19475.276} C_VEL
LIN {X 0,Y 404.397,Z 930.715,A -85,B 0,C 180,E1 19474.858,E2 19474.858} C_VEL
LIN {X 0,Y 399.038,Z 1014.652,A -85,B 0,C 180,E1 19472.38,E2 19472.38} C_VEL
LIN {X 0,Y 396.277,Z 1066.089,A -85,B 0,C 180,E1 19470.664,E2 19470.664} C_VEL
LIN {X 0,Y 395.385,Z 1082.954,A -85,B 0,C 180,E1 19469.881,E2 19469.881} C_VEL
LIN {X 0,Y 394.184,Z 1099.799,A -85,B 0,C 180,E1 19468.813,E2 19468.813} C_VEL
LIN {X 0,Y 392.795,Z 1115.516,A -85,B 0,C 180,E1 19467.518,E2 19467.518} C_VEL
LIN {X 0,Y 391.38,Z 1130.322,A -85,B 0,C 180,E1 19465.986,E2 19465.986} C_VEL
LIN {X 0,Y 389.884,Z 1144.463,A -85,B 0,C 180,E1 19464.145,E2 19464.145} C_VEL
LIN {X 0,Y 388.599,Z 1156.391,A -85,B 0,C 180,E1 19462.225,E2 19462.225} C_VEL
LIN {X 0,Y 387.479,Z 1167.216,A -85,B 0,C 180,E1 19460.072,E2 19460.072} C_VEL
LIN {X 0,Y 386.649,Z 1176.365,A -85,B 0,C 180,E1 19457.767,E2 19457.767} C_VEL
LIN {X 0,Y 386.146,Z 1183.519,A -85,B 0,C 180,E1 19455.469,E2 19455.469} C_VEL
LIN {X 0,Y 385.927,Z 1189.397,A -85,B 0,C 180,E1 19452.875,E2 19452.875} C_VEL
LIN {X 0,Y 386.018,Z 1193.093,A -85,B 0,C 180,E1 19450.447,E2 19450.447} C_VEL
LIN {X 0,Y 386.471,Z 1195.235,A -85,B 0,C 180,E1 19447.732,E2 19447.732} C_VEL
LIN {X 0,Y 387.29,Z 1195.361,A -85,B 0,C 180,E1 19445.184,E2 19445.184} C_VEL
LIN {X 0,Y 388.554,Z 1193.756,A -85,B 0,C 180,E1 19442.655,E2 19442.655} C_VEL
LIN {X 0,Y 390.449,Z 1190.059,A -85,B 0,C 180,E1 19440,E2 19440} C_VEL
LIN {X 0,Y 392.675,Z 1185.049,A -85,B 0,C 180,E1 19437.665,E2 19437.665} C_VEL
LIN {X 0,Y 395.62,Z 1177.704,A -85,B 0,C 180,E1 19435.216,E2 19435.216} C_VEL
LIN {X 0,Y 398.724,Z 1169.348,A -85,B 0,C 180,E1 19433.086,E2 19433.086} C_VEL
LIN {X 0,Y 402.057,Z 1159.7,A -85,B 0,C 180,E1 19431.13,E2 19431.13} C_VEL
LIN {X 0,Y 406.085,Z 1146.879,A -85,B 0,C 180,E1 19429.071,E2 19429.071} C_VEL
LIN {X 0,Y 409.888,Z 1133.361,A -85,B 0,C 180,E1 19427.348,E2 19427.348} C_VEL
LIN {X 0,Y 413.547,Z 1118.761,A -85,B 0,C 180,E1 19425.865,E2 19425.865} C_VEL
LIN {X 0,Y 416.88,Z 1103.619,A -85,B 0,C 180,E1 19424.631,E2 19424.631} C_VEL
LIN {X 0,Y 419.822,Z 1087.563,A -85,B 0,C 180,E1 19423.606,E2 19423.606} C_VEL
LIN {X 0,Y 425.743,Z 1056.799,A -85,B 0,C 180,E1 19422.013,E2 19422.013} C_VEL
LIN {X 0,Y 434.737,Z 1013.64,A -85,B 0,C 180,E1 19420.161,E2 19420.161} C_VEL
LIN {X 0,Y 442.136,Z 974.017,A -85,B 0,C 180,E1 19418.719,E2 19418.719} C_VEL
LIN {X 0,Y 445.37,Z 954.149,A -85,B 0,C 180,E1 19418.049,E2 19418.049} C_VEL
LIN {X 0,Y 445.35,Z 947.843,A -85,B 0,C 180,E1 19417.562,E2 19417.562} C_VEL
LIN {X 0,Y 458.522,Z 915.823,A -85,B 0,C 180,E1 19413.725,E2 19413.725} C_VEL
LIN {X 0,Y 472.943,Z 887.34,A -85,B 0,C 180,E1 19410.209,E2 19410.209} C_VEL
LIN {X 0,Y 488.165,Z 862.838,A -85,B 0,C 180,E1 19407.099,E2 19407.099} C_VEL
LIN {X 0,Y 475.671,Z 882.572,A -85,B 0,C 180,E1 19404.832,E2 19404.832} C_VEL
LIN {X 0,Y 466.191,Z 901.269,A -85,B 0,C 180,E1 19402.474,E2 19402.474} C_VEL
LIN {X 0,Y 459.834,Z 918.436,A -85,B 0,C 180,E1 19400.134,E2 19400.134} C_VEL
LIN {X 0,Y 455.91,Z 936.125,A -85,B 0,C 180,E1 19397.549,E2 19397.549} C_VEL
LIN {X 0,Y 454.874,Z 952.382,A -85,B 0,C 180,E1 19395.054,E2 19395.054} C_VEL
LIN {X 0,Y 455.565,Z 962.141,A -85,B 0,C 180,E1 19393.518,E2 19393.518} C_VEL
LIN {X 0,Y 444.393,Z 984.824,A -85,B 0,C 180,E1 19392.457,E2 19392.457} C_VEL
LIN {X 0,Y 440.476,Z 1009.678,A -85,B 0,C 180,E1 19392.048,E2 19392.048} C_VEL
LIN {X 0,Y 436.889,Z 1031.382,A -85,B 0,C 180,E1 19391.602,E2 19391.602} C_VEL
LIN {X 0,Y 432.323,Z 1057.841,A -85,B 0,C 180,E1 19390.706,E2 19390.706} C_VEL
LIN {X 0,Y 427.526,Z 1081.303,A -85,B 0,C 180,E1 19389.676,E2 19389.676} C_VEL
LIN {X 0,Y 421.899,Z 1106.087,A -85,B 0,C 180,E1 19388.295,E2 19388.295} C_VEL
LIN {X 0,Y 416.188,Z 1129.598,A -85,B 0,C 180,E1 19386.636,E2 19386.636} C_VEL
LIN {X 0,Y 410.968,Z 1150.324,A -85,B 0,C 180,E1 19384.87,E2 19384.87} C_VEL
LIN {X 0,Y 405.627,Z 1170.912,A -85,B 0,C 180,E1 19382.754,E2 19382.754} C_VEL
LIN {X 0,Y 400.577,Z 1190.313,A -85,B 0,C 180,E1 19380.359,E2 19380.359} C_VEL
LIN {X 0,Y 396.209,Z 1207.499,A -85,B 0,C 180,E1 19377.829,E2 19377.829} C_VEL
LIN {X 0,Y 392.159,Z 1224.233,A -85,B 0,C 180,E1 19374.876,E2 19374.876} C_VEL
LIN {X 0,Y 389.417,Z 1237.662,A -85,B 0,C 180,E1 19372.173,E2 19372.173} C_VEL
LIN {X 0,Y 387.482,Z 1250.144,A -85,B 0,C 180,E1 19369.598,E2 19369.598} C_VEL
LIN {X 0,Y 385.944,Z 1261.931,A -85,B 0,C 180,E1 19366.71,E2 19366.71} C_VEL
LIN {X 0,Y 384.993,Z 1271.223,A -85,B 0,C 180,E1 19363.975,E2 19363.975} C_VEL
LIN {X 0,Y 384.446,Z 1279.049,A -85,B 0,C 180,E1 19361.094,E2 19361.094} C_VEL
LIN {X 0,Y 384.265,Z 1285.449,A -85,B 0,C 180,E1 19358.075,E2 19358.075} C_VEL
LIN {X 0,Y 384.28,Z 1289.909,A -85,B 0,C 180,E1 19355.223,E2 19355.223} C_VEL
LIN {X 0,Y 384.344,Z 1292.659,A -85,B 0,C 180,E1 19352.384,E2 19352.384} C_VEL
LIN {X 0,Y 384.336,Z 1293.993,A -85,B 0,C 180,E1 19349.551,E2 19349.551} C_VEL
LIN {X 0,Y 384.25,Z 1293.783,A -85,B 0,C 180,E1 19346.865,E2 19346.865} C_VEL
LIN {X 0,Y 384.145,Z 1292.092,A -85,B 0,C 180,E1 19343.872,E2 19343.872} C_VEL
LIN {X 0,Y 384.209,Z 1288.747,A -85,B 0,C 180,E1 19340.864,E2 19340.864} C_VEL
LIN {X 0,Y 384.679,Z 1283.515,A -85,B 0,C 180,E1 19337.692,E2 19337.692} C_VEL
LIN {X 0,Y 385.757,Z 1276.515,A -85,B 0,C 180,E1 19334.514,E2 19334.514} C_VEL
LIN {X 0,Y 387.608,Z 1267.585,A -85,B 0,C 180,E1 19331.343,E2 19331.343} C_VEL
LIN {X 0,Y 390.189,Z 1257.173,A -85,B 0,C 180,E1 19328.344,E2 19328.344} C_VEL
LIN {X 0,Y 393.861,Z 1244.17,A -85,B 0,C 180,E1 19325.234,E2 19325.234} C_VEL
LIN {X 0,Y 398.374,Z 1229.589,A -85,B 0,C 180,E1 19322.331,E2 19322.331} C_VEL
LIN {X 0,Y 403.601,Z 1213.567,A -85,B 0,C 180,E1 19319.641,E2 19319.641} C_VEL
LIN {X 0,Y 409.862,Z 1195.12,A -85,B 0,C 180,E1 19317.04,E2 19317.04} C_VEL
LIN {X 0,Y 416.878,Z 1174.782,A -85,B 0,C 180,E1 19314.637,E2 19314.637} C_VEL
LIN {X 0,Y 424.507,Z 1152.965,A -85,B 0,C 180,E1 19312.49,E2 19312.49} C_VEL
LIN {X 0,Y 432.59,Z 1129.963,A -85,B 0,C 180,E1 19310.617,E2 19310.617} C_VEL
LIN {X 0,Y 440.538,Z 1107.022,A -85,B 0,C 180,E1 19309.093,E2 19309.093} C_VEL
LIN {X 0,Y 448.44,Z 1083.495,A -85,B 0,C 180,E1 19307.843,E2 19307.843} C_VEL
LIN {X 0,Y 456.406,Z 1058.133,A -85,B 0,C 180,E1 19306.793,E2 19306.793} C_VEL
LIN {X 0,Y 463.105,Z 1034.289,A -85,B 0,C 180,E1 19306.028,E2 19306.028} C_VEL
